LIN {X 0,Y 246.152,Z 600.24,A -85,B 0,C 180,E1 -19920.091,E2 -19920.091} C_VEL
LIN {X 0,Y 247.15,Z 576.037,A -85,B 0,C 180,E1 -19920.831,E2 -19920.831} C_VEL
LIN {X 0,Y 248.137,Z 547.926,A -85,B 0,C 180,E1 -19921.626,E2 -19921.626} C_VEL
LIN {X 0,Y 244.245,Z 525.026,A -85,B 0,C 180,E1 -19922.967,E2 -19922.967} C_VEL
LIN {X 0,Y 243.144,Z 521.008,A -85,B 0,C 180,E1 -19923.272,E2 -19923.272} C_VEL
LIN {X 0,Y 237.077,Z 506.902,A -85,B 0,C 180,E1 -19924.739,E2 -19924.739} C_VEL
LIN {X 0,Y 231.234,Z 495.155,A -85,B 0,C 180,E1 -19926.183,E2 -19926.183} C_VEL
LIN {X 0,Y 230.085,Z 492.253,A -85,B 0,C 180,E1 -19926.602,E2 -19926.602} C_VEL
LIN {X 0,Y 228.669,Z 486.217,A -85,B 0,C 180,E1 -19930.197,E2 -19930.197} C_VEL
LIN {X 0,Y 227.823,Z 482.666,A -85,B 0,C 180,E1 -19932.575,E2 -19932.575} C_VEL
LIN {X 0,Y 227.795,Z 482.606,A -85,B 0,C 180,E1 -19937.251,E2 -19937.251} C_VEL
LIN {X 0,Y 227.844,Z 482.598,A -85,B 0,C 180,E1 -19941.906,E2 -19941.906} C_VEL
LIN {X 0,Y 227.879,Z 482.572,A -85,B 0,C 180,E1 -19946.376,E2 -19946.376} C_VEL
LIN {X 0,Y 227.877,Z 482.596,A -85,B 0,C 180,E1 -19950.429,E2 -19950.429} C_VEL
LIN {X 0,Y 227.867,Z 482.569,A -85,B 0,C 180,E1 -19954.416,E2 -19954.416} C_VEL
LIN {X 0,Y 227.919,Z 482.587,A -85,B 0,C 180,E1 -19958.28,E2 -19958.28} C_VEL
LIN {X 0,Y 227.998,Z 482.563,A -85,B 0,C 180,E1 -19963.891,E2 -19963.891} C_VEL
LIN {X 0,Y 228.123,Z 482.528,A -85,B 0,C 180,E1 -19969.345,E2 -19969.345} C_VEL
LIN {X 0,Y 228.291,Z 482.521,A -85,B 0,C 180,E1 -19972.924,E2 -19972.924} C_VEL
LIN {X 0,Y 228.528,Z 482.492,A -85,B 0,C 180,E1 -19978.235,E2 -19978.235} C_VEL
LIN {X 0,Y 228.503,Z 482.481,A -85,B 0,C 180,E1 -19981.76,E2 -19981.76} C_VEL
LIN {X 0,Y 228.294,Z 482.536,A -85,B 0,C 180,E1 -19987.071,E2 -19987.071} C_VEL
LIN {X 0,Y 228.121,Z 482.525,A -85,B 0,C 180,E1 -19990.649,E2 -19990.649} C_VEL
LIN {X 0,Y 228.004,Z 482.577,A -85,B 0,C 180,E1 -19996.103,E2 -19996.103} C_VEL
LIN {X 0,Y 227.912,Z 482.579,A -85,B 0,C 180,E1 -20001.715,E2 -20001.715} C_VEL
LIN {X 0,Y 227.862,Z 482.571,A -85,B 0,C 180,E1 -20006.563,E2 -20006.563} C_VEL
LIN {X 0,Y 227.861,Z 482.597,A -85,B 0,C 180,E1 -20010.276,E2 -20010.276} C_VEL
LIN {X 0,Y 227.863,Z 482.578,A -85,B 0,C 180,E1 -20013.719,E2 -20013.719} C_VEL
LIN {X 0,Y 227.827,Z 482.608,A -85,B 0,C 180,E1 -20018.09,E2 -20018.09} C_VEL
LIN {X 0,Y 227.772,Z 482.608,A -85,B 0,C 180,E1 -20022.747,E2 -20022.747} C_VEL
LIN {X 0,Y 227.794,Z 482.578,A -85,B 0,C 180,E1 -20025.198,E2 -20025.198} C_VEL
LIN {X 0,Y 227.783,Z 482.557,A -85,B 0,C 180,E1 -20029.615,E2 -20029.615} C_VEL
LIN {X 0,Y 227.873,Z 482.738,A -85,B 0,C 180,E1 -20032.789,E2 -20032.789} C_VEL
LIN {X 0,Y 228.097,Z 483.675,A -85,B 0,C 180,E1 -20033.156,E2 -20033.156} C_VEL
LIN {X 0,Y 229.658,Z 486.481,A -85,B 0,C 180,E1 -20033.59,E2 -20033.59} C_VEL
LIN {X 0,Y 235.192,Z 495.686,A -85,B 0,C 180,E1 -20034.923,E2 -20034.923} C_VEL
LIN {X 0,Y 242.911,Z 509.793,A -85,B 0,C 180,E1 -20036.692,E2 -20036.692} C_VEL
LIN {X 0,Y 251.381,Z 526.173,A -85,B 0,C 180,E1 -20038.501,E2 -20038.501} C_VEL
LIN {X 0,Y 258.769,Z 537.403,A -85,B 0,C 180,E1 -20039.86,E2 -20039.86} C_VEL
LIN {X 0,Y 266.168,Z 546.904,A -85,B 0,C 180,E1 -20041.076,E2 -20041.076} C_VEL
LIN {X 0,Y 278.31,Z 560.203,A -85,B 0,C 180,E1 -20042.838,E2 -20042.838} C_VEL
LIN {X 0,Y 289.982,Z 571.118,A -85,B 0,C 180,E1 -20044.32,E2 -20044.32} C_VEL
LIN {X 0,Y 299.622,Z 579.319,A -85,B 0,C 180,E1 -20045.452,E2 -20045.452} C_VEL
LIN {X 0,Y 307.537,Z 585.808,A -85,B 0,C 180,E1 -20046.478,E2 -20046.478} C_VEL
LIN {X 0,Y 315.775,Z 592.173,A -85,B 0,C 180,E1 -20047.768,E2 -20047.768} C_VEL
LIN {X 0,Y 323.39,Z 597.842,A -85,B 0,C 180,E1 -20049.138,E2 -20049.138} C_VEL
LIN {X 0,Y 330.86,Z 603.38,A -85,B 0,C 180,E1 -20050.658,E2 -20050.658} C_VEL
LIN {X 0,Y 338.279,Z 608.514,A -85,B 0,C 180,E1 -20052.351,E2 -20052.351} C_VEL
LIN {X 0,Y 344.516,Z 613.086,A -85,B 0,C 180,E1 -20053.974,E2 -20053.974} C_VEL
LIN {X 0,Y 348.895,Z 616.008,A -85,B 0,C 180,E1 -20055.206,E2 -20055.206} C_VEL
LIN {X 0,Y 353.8,Z 618.948,A -85,B 0,C 180,E1 -20056.732,E2 -20056.732} C_VEL
LIN {X 0,Y 357.248,Z 621.232,A -85,B 0,C 180,E1 -20057.965,E2 -20057.965} C_VEL
LIN {X 0,Y 361.911,Z 624.66,A -85,B 0,C 180,E1 -20059.935,E2 -20059.935} C_VEL
LIN {X 0,Y 364.421,Z 626.158,A -85,B 0,C 180,E1 -20061.125,E2 -20061.125} C_VEL
LIN {X 0,Y 368.041,Z 628.101,A -85,B 0,C 180,E1 -20063.184,E2 -20063.184} C_VEL
LIN {X 0,Y 369.955,Z 628.948,A -85,B 0,C 180,E1 -20064.55,E2 -20064.55} C_VEL
LIN {X 0,Y 371.243,Z 629.373,A -85,B 0,C 180,E1 -20065.657,E2 -20065.657} C_VEL
LIN {X 0,Y 372.23,Z 629.672,A -85,B 0,C 180,E1 -20066.753,E2 -20066.753} C_VEL
LIN {X 0,Y 372.855,Z 630.069,A -85,B 0,C 180,E1 -20067.84,E2 -20067.84} C_VEL
LIN {X 0,Y 373.209,Z 630.352,A -85,B 0,C 180,E1 -20068.921,E2 -20068.921} C_VEL
LIN {X 0,Y 373.398,Z 630.248,A -85,B 0,C 180,E1 -20070,E2 -20070} C_VEL
LIN {X 0,Y 373.231,Z 630.289,A -85,B 0,C 180,E1 -20071.079,E2 -20071.079} C_VEL
LIN {X 0,Y 372.781,Z 630.004,A -85,B 0,C 180,E1 -20072.349,E2 -20072.349} C_VEL
LIN {X 0,Y 372.229,Z 629.672,A -85,B 0,C 180,E1 -20073.247,E2 -20073.247} C_VEL
LIN {X 0,Y 371.24,Z 629.386,A -85,B 0,C 180,E1 -20074.343,E2 -20074.343} C_VEL
LIN {X 0,Y 369.963,Z 628.952,A -85,B 0,C 180,E1 -20075.45,E2 -20075.45} C_VEL
LIN {X 0,Y 368.049,Z 628.078,A -85,B 0,C 180,E1 -20076.826,E2 -20076.826} C_VEL
LIN {X 0,Y 366.561,Z 627.405,A -85,B 0,C 180,E1 -20077.713,E2 -20077.713} C_VEL
LIN {X 0,Y 363.297,Z 625.502,A -85,B 0,C 180,E1 -20079.407,E2 -20079.407} C_VEL
LIN {X 0,Y 361.921,Z 624.674,A -85,B 0,C 180,E1 -20080.065,E2 -20080.065} C_VEL
LIN {X 0,Y 357.616,Z 621.526,A -85,B 0,C 180,E1 -20081.887,E2 -20081.887} C_VEL
LIN {X 0,Y 353.791,Z 618.959,A -85,B 0,C 180,E1 -20083.262,E2 -20083.262} C_VEL
LIN {X 0,Y 347.291,Z 614.974,A -85,B 0,C 180,E1 -20085.252,E2 -20085.252} C_VEL
LIN {X 0,Y 340.677,Z 610.221,A -85,B 0,C 180,E1 -20087.062,E2 -20087.062} C_VEL
LIN {X 0,Y 333.125,Z 605.057,A -85,B 0,C 180,E1 -20088.843,E2 -20088.843} C_VEL
LIN {X 0,Y 324.559,Z 598.647,A -85,B 0,C 180,E1 -20090.638,E2 -20090.638} C_VEL
LIN {X 0,Y 316.695,Z 592.953,A -85,B 0,C 180,E1 -20092.071,E2 -20092.071} C_VEL
LIN {X 0,Y 308.97,Z 586.887,A -85,B 0,C 180,E1 -20093.315,E2 -20093.315} C_VEL
LIN {X 0,Y 301.688,Z 581.017,A -85,B 0,C 180,E1 -20094.302,E2 -20094.302} C_VEL
LIN {X 0,Y 290.907,Z 571.969,A -85,B 0,C 180,E1 -20095.569,E2 -20095.569} C_VEL
LIN {X 0,Y 280.514,Z 562.3,A -85,B 0,C 180,E1 -20096.87,E2 -20096.87} C_VEL
LIN {X 0,Y 268.243,Z 549.356,A -85,B 0,C 180,E1 -20098.604,E2 -20098.604} C_VEL
LIN {X 0,Y 260.21,Z 539.392,A -85,B 0,C 180,E1 -20099.892,E2 -20099.892} C_VEL
LIN {X 0,Y 251.95,Z 527.134,A -85,B 0,C 180,E1 -20101.388,E2 -20101.388} C_VEL
LIN {X 0,Y 244.918,Z 513.819,A -85,B 0,C 180,E1 -20102.86,E2 -20102.86} C_VEL
LIN {X 0,Y 237.684,Z 500.018,A -85,B 0,C 180,E1 -20104.497,E2 -20104.497} C_VEL
LIN {X 0,Y 231.453,Z 489.468,A -85,B 0,C 180,E1 -20105.968,E2 -20105.968} C_VEL
LIN {X 0,Y 229.657,Z 486.509,A -85,B 0,C 180,E1 -20106.409,E2 -20106.409} C_VEL
LIN {X 0,Y 228.093,Z 483.698,A -85,B 0,C 180,E1 -20106.843,E2 -20106.843} C_VEL
LIN {X 0,Y 227.873,Z 482.743,A -85,B 0,C 180,E1 -20107.212,E2 -20107.212} C_VEL
LIN {X 0,Y 227.783,Z 482.557,A -85,B 0,C 180,E1 -20110.385,E2 -20110.385} C_VEL
LIN {X 0,Y 227.795,Z 482.588,A -85,B 0,C 180,E1 -20115.202,E2 -20115.202} C_VEL
LIN {X 0,Y 227.786,Z 482.59,A -85,B 0,C 180,E1 -20119.619,E2 -20119.619} C_VEL
LIN {X 0,Y 227.849,Z 482.584,A -85,B 0,C 180,E1 -20124.126,E2 -20124.126} C_VEL
LIN {X 0,Y 227.845,Z 482.605,A -85,B 0,C 180,E1 -20128.378,E2 -20128.378} C_VEL
LIN {X 0,Y 227.825,Z 482.572,A -85,B 0,C 180,E1 -20132.44,E2 -20132.44} C_VEL
LIN {X 0,Y 227.858,Z 482.603,A -85,B 0,C 180,E1 -20136.365,E2 -20136.365} C_VEL
LIN {X 0,Y 227.88,Z 482.559,A -85,B 0,C 180,E1 -20140.172,E2 -20140.172} C_VEL
LIN {X 0,Y 228.004,Z 482.577,A -85,B 0,C 180,E1 -20143.897,E2 -20143.897} C_VEL
LIN {X 0,Y 228.121,Z 482.525,A -85,B 0,C 180,E1 -20149.351,E2 -20149.351} C_VEL
LIN {X 0,Y 228.294,Z 482.536,A -85,B 0,C 180,E1 -20152.929,E2 -20152.929} C_VEL
LIN {X 0,Y 228.503,Z 482.481,A -85,B 0,C 180,E1 -20158.24,E2 -20158.24} C_VEL
LIN {X 0,Y 228.528,Z 482.492,A -85,B 0,C 180,E1 -20161.765,E2 -20161.765} C_VEL
LIN {X 0,Y 228.291,Z 482.521,A -85,B 0,C 180,E1 -20167.076,E2 -20167.076} C_VEL
LIN {X 0,Y 228.123,Z 482.528,A -85,B 0,C 180,E1 -20170.655,E2 -20170.655} C_VEL
LIN {X 0,Y 227.998,Z 482.563,A -85,B 0,C 180,E1 -20176.109,E2 -20176.109} C_VEL
LIN {X 0,Y 227.919,Z 482.587,A -85,B 0,C 180,E1 -20181.72,E2 -20181.72} C_VEL
LIN {X 0,Y 227.872,Z 482.564,A -85,B 0,C 180,E1 -20186.568,E2 -20186.568} C_VEL
LIN {X 0,Y 227.875,Z 482.601,A -85,B 0,C 180,E1 -20190.282,E2 -20190.282} C_VEL
LIN {X 0,Y 227.876,Z 482.572,A -85,B 0,C 180,E1 -20193.723,E2 -20193.723} C_VEL
LIN {X 0,Y 227.844,Z 482.598,A -85,B 0,C 180,E1 -20198.094,E2 -20198.094} C_VEL
LIN {X 0,Y 227.795,Z 482.606,A -85,B 0,C 180,E1 -20202.749,E2 -20202.749} C_VEL
LIN {X 0,Y 227.821,Z 482.677,A -85,B 0,C 180,E1 -20207.425,E2 -20207.425} C_VEL
LIN {X 0,Y 229.242,Z 488.495,A -85,B 0,C 180,E1 -20211.232,E2 -20211.232} C_VEL
LIN {X 0,Y 230.107,Z 492.26,A -85,B 0,C 180,E1 -20213.403,E2 -20213.403} C_VEL
LIN {X 0,Y 231.786,Z 496.084,A -85,B 0,C 180,E1 -20213.951,E2 -20213.951} C_VEL
LIN {X 0,Y 238.336,Z 509.677,A -85,B 0,C 180,E1 -20215.568,E2 -20215.568} C_VEL
LIN {X 0,Y 243.688,Z 522.323,A -85,B 0,C 180,E1 -20216.856,E2 -20216.856} C_VEL
LIN {X 0,Y 247.536,Z 543.646,A -85,B 0,C 180,E1 -20218.146,E2 -20218.146} C_VEL
LIN {X 0,Y 248.135,Z 549.551,A -85,B 0,C 180,E1 -20218.428,E2 -20218.428} C_VEL
LIN {X 0,Y 248.055,Z 551.394,A -85,B 0,C 180,E1 -20218.478,E2 -20218.478} C_VEL
LIN {X 0,Y 247.294,Z 555.318,A -85,B 0,C 180,E1 -20218.501,E2 -20218.501} C_VEL
LIN {X 0,Y 241.893,Z 567.619,A -85,B 0,C 180,E1 -20218.141,E2 -20218.141} C_VEL
LIN {X 0,Y 241.238,Z 571.533,A -85,B 0,C 180,E1 -20218.179,E2 -20218.179} C_VEL
LIN {X 0,Y 240.016,Z 599.524,A -85,B 0,C 180,E1 -20219.032,E2 -20219.032} C_VEL
LIN {X 0,Y 239.072,Z 609.938,A -85,B 0,C 180,E1 -20219.538,E2 -20219.538} C_VEL
LIN {X 0,Y 237.776,Z 619.744,A -85,B 0,C 180,E1 -20220.203,E2 -20220.203} C_VEL
LIN {X 0,Y 236.276,Z 629.543,A -85,B 0,C 180,E1 -20221.096,E2 -20221.096} C_VEL
LIN {X 0,Y 234.598,Z 638.308,A -85,B 0,C 180,E1 -20222.09,E2 -20222.09} C_VEL
LIN {X 0,Y 232.712,Z 647.03,A -85,B 0,C 180,E1 -20223.306,E2 -20223.306} C_VEL
LIN {X 0,Y 230.942,Z 654.441,A -85,B 0,C 180,E1 -20224.542,E2 -20224.542} C_VEL
LIN {X 0,Y 229.022,Z 661.859,A -85,B 0,C 180,E1 -20226.009,E2 -20226.009} C_VEL
LIN {X 0,Y 227.089,Z 669.094,A -85,B 0,C 180,E1 -20227.721,E2 -20227.721} C_VEL
LIN {X 0,Y 225.118,Z 676.649,A -85,B 0,C 180,E1 -20229.915,E2 -20229.915} C_VEL
LIN {X 0,Y 223.195,Z 682.958,A -85,B 0,C 180,E1 -20232.121,E2 -20232.121} C_VEL
LIN {X 0,Y 221.66,Z 688.231,A -85,B 0,C 180,E1 -20234.366,E2 -20234.366} C_VEL
LIN {X 0,Y 220.23,Z 693.327,A -85,B 0,C 180,E1 -20237.092,E2 -20237.092} C_VEL
LIN {X 0,Y 219.325,Z 697.296,A -85,B 0,C 180,E1 -20239.849,E2 -20239.849} C_VEL
LIN {X 0,Y 218.716,Z 700.234,A -85,B 0,C 180,E1 -20242.615,E2 -20242.615} C_VEL
LIN {X 0,Y 218.512,Z 701.738,A -85,B 0,C 180,E1 -20244.463,E2 -20244.463} C_VEL
LIN {X 0,Y 218.526,Z 703.271,A -85,B 0,C 180,E1 -20248.157,E2 -20248.157} C_VEL
LIN {X 0,Y 218.625,Z 703.554,A -85,B 0,C 180,E1 -20250,E2 -20250} C_VEL
LIN {X 0,Y 218.506,Z 702.672,A -85,B 0,C 180,E1 -20253.688,E2 -20253.688} C_VEL
LIN {X 0,Y 218.572,Z 701.74,A -85,B 0,C 180,E1 -20255.535,E2 -20255.535} C_VEL
LIN {X 0,Y 219.094,Z 698.386,A -85,B 0,C 180,E1 -20259.229,E2 -20259.229} C_VEL
LIN {X 0,Y 219.886,Z 694.756,A -85,B 0,C 180,E1 -20261.991,E2 -20261.991} C_VEL
LIN {X 0,Y 221.084,Z 690.02,A -85,B 0,C 180,E1 -20264.733,E2 -20264.733} C_VEL
LIN {X 0,Y 222.92,Z 684.052,A -85,B 0,C 180,E1 -20267.428,E2 -20267.428} C_VEL
LIN {X 0,Y 224.301,Z 679.271,A -85,B 0,C 180,E1 -20269.208,E2 -20269.208} C_VEL
LIN {X 0,Y 226.061,Z 673.153,A -85,B 0,C 180,E1 -20271.14,E2 -20271.14} C_VEL
LIN {X 0,Y 228.034,Z 665.56,A -85,B 0,C 180,E1 -20273.138,E2 -20273.138} C_VEL
LIN {X 0,Y 230.131,Z 657.736,A -85,B 0,C 180,E1 -20274.829,E2 -20274.829} C_VEL
LIN {X 0,Y 232.108,Z 649.654,A -85,B 0,C 180,E1 -20276.284,E2 -20276.284} C_VEL
LIN {X 0,Y 234.303,Z 639.898,A -85,B 0,C 180,E1 -20277.705,E2 -20277.705} C_VEL
LIN {X 0,Y 235.954,Z 631.511,A -85,B 0,C 180,E1 -20278.704,E2 -20278.704} C_VEL
LIN {X 0,Y 237.557,Z 621.005,A -85,B 0,C 180,E1 -20279.705,E2 -20279.705} C_VEL
LIN {X 0,Y 238.961,Z 610.702,A -85,B 0,C 180,E1 -20280.423,E2 -20280.423} C_VEL
LIN {X 0,Y 239.98,Z 600.72,A -85,B 0,C 180,E1 -20280.917,E2 -20280.917} C_VEL
LIN {X 0,Y 240.951,Z 579.375,A -85,B 0,C 180,E1 -20281.594,E2 -20281.594} C_VEL
LIN {X 0,Y 241.993,Z 548.404,A -85,B 0,C 180,E1 -20282.503,E2 -20282.503} C_VEL
LIN {X 0,Y 238.141,Z 525.634,A -85,B 0,C 180,E1 -20283.896,E2 -20283.896} C_VEL
LIN {X 0,Y 232.971,Z 512.992,A -85,B 0,C 180,E1 -20285.213,E2 -20285.213} C_VEL
LIN {X 0,Y 226.478,Z 499.636,A -85,B 0,C 180,E1 -20286.888,E2 -20286.888} C_VEL
LIN {X 0,Y 223.937,Z 494.745,A -85,B 0,C 180,E1 -20287.567,E2 -20287.567} C_VEL
LIN {X 0,Y 222.807,Z 492.019,A -85,B 0,C 180,E1 -20288.001,E2 -20288.001} C_VEL
LIN {X 0,Y 221.315,Z 485.957,A -85,B 0,C 180,E1 -20291.825,E2 -20291.825} C_VEL
LIN {X 0,Y 220.753,Z 483.553,A -85,B 0,C 180,E1 -20293.585,E2 -20293.585} C_VEL
LIN {X 0,Y 220.756,Z 483.487,A -85,B 0,C 180,E1 -20298.041,E2 -20298.041} C_VEL
LIN {X 0,Y 220.829,Z 483.479,A -85,B 0,C 180,E1 -20302.791,E2 -20302.791} C_VEL
LIN {X 0,Y 220.814,Z 483.457,A -85,B 0,C 180,E1 -20307.241,E2 -20307.241} C_VEL
LIN {X 0,Y 220.796,Z 483.46,A -85,B 0,C 180,E1 -20311.478,E2 -20311.478} C_VEL
LIN {X 0,Y 220.797,Z 483.464,A -85,B 0,C 180,E1 -20315.554,E2 -20315.554} C_VEL
LIN {X 0,Y 220.845,Z 483.449,A -85,B 0,C 180,E1 -20319.507,E2 -20319.507} C_VEL
LIN {X 0,Y 220.944,Z 483.431,A -85,B 0,C 180,E1 -20323.362,E2 -20323.362} C_VEL
LIN {X 0,Y 221.045,Z 483.413,A -85,B 0,C 180,E1 -20329,E2 -20329} C_VEL
LIN {X 0,Y 221.228,Z 483.396,A -85,B 0,C 180,E1 -20332.697,E2 -20332.697} C_VEL
LIN {X 0,Y 221.461,Z 483.372,A -85,B 0,C 180,E1 -20338.179,E2 -20338.179} C_VEL
LIN {X 0,Y 221.538,Z 483.341,A -85,B 0,C 180,E1 -20339.997,E2 -20339.997} C_VEL
LIN {X 0,Y 221.441,Z 483.36,A -85,B 0,C 180,E1 -20341.816,E2 -20341.816} C_VEL
LIN {X 0,Y 221.231,Z 483.411,A -85,B 0,C 180,E1 -20347.297,E2 -20347.297} C_VEL
LIN {X 0,Y 221.046,Z 483.407,A -85,B 0,C 180,E1 -20350.994,E2 -20350.994} C_VEL
LIN {X 0,Y 220.964,Z 483.446,A -85,B 0,C 180,E1 -20356.631,E2 -20356.631} C_VEL
LIN {X 0,Y 220.838,Z 483.44,A -85,B 0,C 180,E1 -20360.488,E2 -20360.488} C_VEL
LIN {X 0,Y 220.796,Z 483.478,A -85,B 0,C 180,E1 -20364.44,E2 -20364.44} C_VEL
LIN {X 0,Y 220.784,Z 483.453,A -85,B 0,C 180,E1 -20368.517,E2 -20368.517} C_VEL
LIN {X 0,Y 220.801,Z 483.468,A -85,B 0,C 180,E1 -20372.755,E2 -20372.755} C_VEL
LIN {X 0,Y 220.787,Z 483.483,A -85,B 0,C 180,E1 -20377.271,E2 -20377.271} C_VEL
LIN {X 0,Y 220.734,Z 483.474,A -85,B 0,C 180,E1 -20381.956,E2 -20381.956} C_VEL
LIN {X 0,Y 220.737,Z 483.447,A -85,B 0,C 180,E1 -20385.537,E2 -20385.537} C_VEL
LIN {X 0,Y 220.767,Z 483.444,A -85,B 0,C 180,E1 -20390.455,E2 -20390.455} C_VEL
LIN {X 0,Y 220.819,Z 483.766,A -85,B 0,C 180,E1 -20391.531,E2 -20391.531} C_VEL
LIN {X 0,Y 221.111,Z 484.873,A -85,B 0,C 180,E1 -20391.844,E2 -20391.844} C_VEL
LIN {X 0,Y 222.659,Z 487.488,A -85,B 0,C 180,E1 -20392.28,E2 -20392.28} C_VEL
LIN {X 0,Y 228.617,Z 497.051,A -85,B 0,C 180,E1 -20393.801,E2 -20393.801} C_VEL
LIN {X 0,Y 236.784,Z 511.74,A -85,B 0,C 180,E1 -20395.775,E2 -20395.775} C_VEL
LIN {X 0,Y 246.092,Z 530.036,A -85,B 0,C 180,E1 -20397.868,E2 -20397.868} C_VEL
LIN {X 0,Y 253.652,Z 541.708,A -85,B 0,C 180,E1 -20399.32,E2 -20399.32} C_VEL
LIN {X 0,Y 261.138,Z 551.49,A -85,B 0,C 180,E1 -20400.601,E2 -20400.601} C_VEL
LIN {X 0,Y 273.853,Z 565.494,A -85,B 0,C 180,E1 -20402.508,E2 -20402.508} C_VEL
LIN {X 0,Y 285.738,Z 576.669,A -85,B 0,C 180,E1 -20404.058,E2 -20404.058} C_VEL
LIN {X 0,Y 297.612,Z 586.737,A -85,B 0,C 180,E1 -20405.485,E2 -20405.485} C_VEL
LIN {X 0,Y 306.322,Z 593.716,A -85,B 0,C 180,E1 -20406.682,E2 -20406.682} C_VEL
LIN {X 0,Y 315.161,Z 600.552,A -85,B 0,C 180,E1 -20408.13,E2 -20408.13} C_VEL
LIN {X 0,Y 323.976,Z 606.917,A -85,B 0,C 180,E1 -20409.785,E2 -20409.785} C_VEL
LIN {X 0,Y 331.811,Z 612.657,A -85,B 0,C 180,E1 -20411.476,E2 -20411.476} C_VEL
LIN {X 0,Y 338.065,Z 616.973,A -85,B 0,C 180,E1 -20412.988,E2 -20412.988} C_VEL
LIN {X 0,Y 343.987,Z 621.179,A -85,B 0,C 180,E1 -20414.597,E2 -20414.597} C_VEL
LIN {X 0,Y 348.69,Z 624.181,A -85,B 0,C 180,E1 -20416.004,E2 -20416.004} C_VEL
LIN {X 0,Y 352.888,Z 626.57,A -85,B 0,C 180,E1 -20417.375,E2 -20417.375} C_VEL
LIN {X 0,Y 357.609,Z 630.137,A -85,B 0,C 180,E1 -20419.294,E2 -20419.294} C_VEL
LIN {X 0,Y 361.372,Z 632.529,A -85,B 0,C 180,E1 -20421.049,E2 -20421.049} C_VEL
LIN {X 0,Y 363.548,Z 633.753,A -85,B 0,C 180,E1 -20422.223,E2 -20422.223} C_VEL
LIN {X 0,Y 365.426,Z 634.705,A -85,B 0,C 180,E1 -20423.374,E2 -20423.374} C_VEL
LIN {X 0,Y 367.09,Z 635.43,A -85,B 0,C 180,E1 -20424.566,E2 -20424.566} C_VEL
LIN {X 0,Y 368.312,Z 635.847,A -85,B 0,C 180,E1 -20425.623,E2 -20425.623} C_VEL
LIN {X 0,Y 369.331,Z 636.134,A -85,B 0,C 180,E1 -20426.727,E2 -20426.727} C_VEL
LIN {X 0,Y 369.963,Z 636.524,A -85,B 0,C 180,E1 -20427.823,E2 -20427.823} C_VEL
LIN {X 0,Y 370.313,Z 636.808,A -85,B 0,C 180,E1 -20428.913,E2 -20428.913} C_VEL
LIN {X 0,Y 370.515,Z 636.708,A -85,B 0,C 180,E1 -20430,E2 -20430} C_VEL
LIN {X 0,Y 370.326,Z 636.764,A -85,B 0,C 180,E1 -20431.087,E2 -20431.087} C_VEL
LIN {X 0,Y 369.952,Z 636.522,A -85,B 0,C 180,E1 -20432.177,E2 -20432.177} C_VEL
LIN {X 0,Y 369.319,Z 636.128,A -85,B 0,C 180,E1 -20433.273,E2 -20433.273} C_VEL
LIN {X 0,Y 368.302,Z 635.842,A -85,B 0,C 180,E1 -20434.378,E2 -20434.378} C_VEL
LIN {X 0,Y 367.004,Z 635.393,A -85,B 0,C 180,E1 -20435.494,E2 -20435.494} C_VEL
LIN {X 0,Y 365.433,Z 634.696,A -85,B 0,C 180,E1 -20436.626,E2 -20436.626} C_VEL
LIN {X 0,Y 362.33,Z 633.119,A -85,B 0,C 180,E1 -20438.433,E2 -20438.433} C_VEL
LIN {X 0,Y 358.825,Z 631.037,A -85,B 0,C 180,E1 -20440.153,E2 -20440.153} C_VEL
LIN {X 0,Y 354.949,Z 628.21,A -85,B 0,C 180,E1 -20441.81,E2 -20441.81} C_VEL
LIN {X 0,Y 350.813,Z 625.364,A -85,B 0,C 180,E1 -20443.331,E2 -20443.331} C_VEL
LIN {X 0,Y 345.964,Z 622.467,A -85,B 0,C 180,E1 -20444.821,E2 -20444.821} C_VEL
LIN {X 0,Y 340.893,Z 619.012,A -85,B 0,C 180,E1 -20446.272,E2 -20446.272} C_VEL
LIN {X 0,Y 335.959,Z 615.335,A -85,B 0,C 180,E1 -20447.558,E2 -20447.558} C_VEL
LIN {X 0,Y 329.273,Z 610.899,A -85,B 0,C 180,E1 -20449.085,E2 -20449.085} C_VEL
LIN {X 0,Y 321.066,Z 604.786,A -85,B 0,C 180,E1 -20450.789,E2 -20450.789} C_VEL
LIN {X 0,Y 312.942,Z 598.863,A -85,B 0,C 180,E1 -20452.252,E2 -20452.252} C_VEL
LIN {X 0,Y 304.378,Z 592.212,A -85,B 0,C 180,E1 -20453.605,E2 -20453.605} C_VEL
LIN {X 0,Y 295.74,Z 585.188,A -85,B 0,C 180,E1 -20454.744,E2 -20454.744} C_VEL
LIN {X 0,Y 281.267,Z 572.743,A -85,B 0,C 180,E1 -20456.499,E2 -20456.499} C_VEL
LIN {X 0,Y 266.835,Z 558.072,A -85,B 0,C 180,E1 -20458.508,E2 -20458.508} C_VEL
LIN {X 0,Y 256.198,Z 545.289,A -85,B 0,C 180,E1 -20460.226,E2 -20460.226} C_VEL
LIN {X 0,Y 247.6,Z 532.566,A -85,B 0,C 180,E1 -20461.826,E2 -20461.826} C_VEL
LIN {X 0,Y 240.523,Z 519.383,A -85,B 0,C 180,E1 -20463.348,E2 -20463.348} C_VEL
LIN {X 0,Y 233.626,Z 505.89,A -85,B 0,C 180,E1 -20464.973,E2 -20464.973} C_VEL
LIN {X 0,Y 226.56,Z 493.674,A -85,B 0,C 180,E1 -20466.714,E2 -20466.714} C_VEL
LIN {X 0,Y 222.66,Z 487.466,A -85,B 0,C 180,E1 -20467.72,E2 -20467.72} C_VEL
LIN {X 0,Y 221.111,Z 484.873,A -85,B 0,C 180,E1 -20468.156,E2 -20468.156} C_VEL
LIN {X 0,Y 220.82,Z 483.706,A -85,B 0,C 180,E1 -20468.517,E2 -20468.517} C_VEL
LIN {X 0,Y 220.728,Z 483.423,A -85,B 0,C 180,E1 -20471.962,E2 -20471.962} C_VEL
LIN {X 0,Y 220.739,Z 483.474,A -85,B 0,C 180,E1 -20475.542,E2 -20475.542} C_VEL
LIN {X 0,Y 220.77,Z 483.469,A -85,B 0,C 180,E1 -20480.459,E2 -20480.459} C_VEL
LIN {X 0,Y 220.816,Z 483.479,A -85,B 0,C 180,E1 -20482.795,E2 -20482.795} C_VEL
LIN {X 0,Y 220.801,Z 483.468,A -85,B 0,C 180,E1 -20487.245,E2 -20487.245} C_VEL
LIN {X 0,Y 220.784,Z 483.453,A -85,B 0,C 180,E1 -20491.483,E2 -20491.483} C_VEL
LIN {X 0,Y 220.796,Z 483.478,A -85,B 0,C 180,E1 -20495.56,E2 -20495.56} C_VEL
LIN {X 0,Y 220.838,Z 483.44,A -85,B 0,C 180,E1 -20499.512,E2 -20499.512} C_VEL
LIN {X 0,Y 220.964,Z 483.446,A -85,B 0,C 180,E1 -20503.369,E2 -20503.369} C_VEL
LIN {X 0,Y 221.046,Z 483.407,A -85,B 0,C 180,E1 -20509.006,E2 -20509.006} C_VEL
LIN {X 0,Y 221.231,Z 483.411,A -85,B 0,C 180,E1 -20512.703,E2 -20512.703} C_VEL
LIN {X 0,Y 221.441,Z 483.36,A -85,B 0,C 180,E1 -20518.184,E2 -20518.184} C_VEL
LIN {X 0,Y 221.538,Z 483.341,A -85,B 0,C 180,E1 -20520.003,E2 -20520.003} C_VEL
LIN {X 0,Y 221.461,Z 483.372,A -85,B 0,C 180,E1 -20521.821,E2 -20521.821} C_VEL
LIN {X 0,Y 221.228,Z 483.396,A -85,B 0,C 180,E1 -20527.303,E2 -20527.303} C_VEL
LIN {X 0,Y 221.045,Z 483.413,A -85,B 0,C 180,E1 -20531,E2 -20531} C_VEL
LIN {X 0,Y 220.944,Z 483.431,A -85,B 0,C 180,E1 -20536.638,E2 -20536.638} C_VEL
LIN {X 0,Y 220.845,Z 483.449,A -85,B 0,C 180,E1 -20540.493,E2 -20540.493} C_VEL
LIN {X 0,Y 220.797,Z 483.464,A -85,B 0,C 180,E1 -20544.446,E2 -20544.446} C_VEL
LIN {X 0,Y 220.796,Z 483.46,A -85,B 0,C 180,E1 -20548.522,E2 -20548.522} C_VEL
LIN {X 0,Y 220.814,Z 483.457,A -85,B 0,C 180,E1 -20552.759,E2 -20552.759} C_VEL
LIN {X 0,Y 220.806,Z 483.482,A -85,B 0,C 180,E1 -20557.277,E2 -20557.277} C_VEL
LIN {X 0,Y 220.756,Z 483.487,A -85,B 0,C 180,E1 -20561.959,E2 -20561.959} C_VEL
LIN {X 0,Y 220.757,Z 483.626,A -85,B 0,C 180,E1 -20566.572,E2 -20566.572} C_VEL
LIN {X 0,Y 222.639,Z 491.302,A -85,B 0,C 180,E1 -20571.655,E2 -20571.655} C_VEL
LIN {X 0,Y 222.985,Z 492.547,A -85,B 0,C 180,E1 -20572.122,E2 -20572.122} C_VEL
LIN {X 0,Y 229.695,Z 506.052,A -85,B 0,C 180,E1 -20573.951,E2 -20573.951} C_VEL
LIN {X 0,Y 236.302,Z 520.801,A -85,B 0,C 180,E1 -20575.633,E2 -20575.633} C_VEL
LIN {X 0,Y 238.277,Z 526.324,A -85,B 0,C 180,E1 -20576.151,E2 -20576.151} C_VEL
LIN {X 0,Y 241.849,Z 547.149,A -85,B 0,C 180,E1 -20577.432,E2 -20577.432} C_VEL
LIN {X 0,Y 242.006,Z 552.1,A -85,B 0,C 180,E1 -20577.626,E2 -20577.626} C_VEL
LIN {X 0,Y 241.238,Z 571.533,A -85,B 0,C 180,E1 -20578.179,E2 -20578.179} C_VEL
LIN {X 0,Y 240.553,Z 577.376,A -85,B 0,C 180,E1 -20578.277,E2 -20578.277} C_VEL
LIN {X 0,Y 237.721,Z 586.874,A -85,B 0,C 180,E1 -20578.19,E2 -20578.19} C_VEL
LIN {X 0,Y 234.727,Z 596.356,A -85,B 0,C 180,E1 -20578.103,E2 -20578.103} C_VEL
LIN {X 0,Y 233.807,Z 602.18,A -85,B 0,C 180,E1 -20578.252,E2 -20578.252} C_VEL
LIN {X 0,Y 232.231,Z 615.762,A -85,B 0,C 180,E1 -20579.038,E2 -20579.038} C_VEL
LIN {X 0,Y 230.818,Z 625.412,A -85,B 0,C 180,E1 -20579.842,E2 -20579.842} C_VEL
LIN {X 0,Y 228.657,Z 636.521,A -85,B 0,C 180,E1 -20581.047,E2 -20581.047} C_VEL
LIN {X 0,Y 226.721,Z 645.521,A -85,B 0,C 180,E1 -20582.292,E2 -20582.292} C_VEL
LIN {X 0,Y 224.518,Z 654.244,A -85,B 0,C 180,E1 -20583.759,E2 -20583.759} C_VEL
LIN {X 0,Y 222.529,Z 661.662,A -85,B 0,C 180,E1 -20585.262,E2 -20585.262} C_VEL
LIN {X 0,Y 220.049,Z 670.458,A -85,B 0,C 180,E1 -20587.464,E2 -20587.464} C_VEL
LIN {X 0,Y 218.421,Z 676.452,A -85,B 0,C 180,E1 -20589.272,E2 -20589.272} C_VEL
LIN {X 0,Y 216.398,Z 682.76,A -85,B 0,C 180,E1 -20591.54,E2 -20591.54} C_VEL
LIN {X 0,Y 214.806,Z 688.034,A -85,B 0,C 180,E1 -20593.853,E2 -20593.853} C_VEL
LIN {X 0,Y 213.266,Z 693.129,A -85,B 0,C 180,E1 -20596.663,E2 -20596.663} C_VEL
LIN {X 0,Y 212.311,Z 697.099,A -85,B 0,C 180,E1 -20599.51,E2 -20599.51} C_VEL
LIN {X 0,Y 211.656,Z 700.038,A -85,B 0,C 180,E1 -20602.368,E2 -20602.368} C_VEL
LIN {X 0,Y 211.44,Z 701.542,A -85,B 0,C 180,E1 -20604.277,E2 -20604.277} C_VEL
LIN {X 0,Y 211.429,Z 703.075,A -85,B 0,C 180,E1 -20608.095,E2 -20608.095} C_VEL
LIN {X 0,Y 211.541,Z 703.358,A -85,B 0,C 180,E1 -20610,E2 -20610} C_VEL
LIN {X 0,Y 211.404,Z 702.475,A -85,B 0,C 180,E1 -20613.812,E2 -20613.812} C_VEL
LIN {X 0,Y 211.494,Z 701.543,A -85,B 0,C 180,E1 -20615.721,E2 -20615.721} C_VEL
LIN {X 0,Y 212.068,Z 698.19,A -85,B 0,C 180,E1 -20619.538,E2 -20619.538} C_VEL
LIN {X 0,Y 212.909,Z 694.559,A -85,B 0,C 180,E1 -20622.39,E2 -20622.39} C_VEL
LIN {X 0,Y 214.209,Z 689.824,A -85,B 0,C 180,E1 -20625.217,E2 -20625.217} C_VEL
LIN {X 0,Y 216.112,Z 683.854,A -85,B 0,C 180,E1 -20627.995,E2 -20627.995} C_VEL
LIN {X 0,Y 217.603,Z 679.075,A -85,B 0,C 180,E1 -20629.823,E2 -20629.823} C_VEL
LIN {X 0,Y 219.429,Z 672.84,A -85,B 0,C 180,E1 -20631.847,E2 -20631.847} C_VEL
LIN {X 0,Y 221.503,Z 665.363,A -85,B 0,C 180,E1 -20633.862,E2 -20633.862} C_VEL
LIN {X 0,Y 223.675,Z 657.539,A -85,B 0,C 180,E1 -20635.596,E2 -20635.596} C_VEL
LIN {X 0,Y 225.757,Z 649.458,A -85,B 0,C 180,E1 -20637.083,E2 -20637.083} C_VEL
LIN {X 0,Y 228.03,Z 639.701,A -85,B 0,C 180,E1 -20638.536,E2 -20638.536} C_VEL
LIN {X 0,Y 229.756,Z 631.315,A -85,B 0,C 180,E1 -20639.554,E2 -20639.554} C_VEL
LIN {X 0,Y 231.42,Z 620.808,A -85,B 0,C 180,E1 -20640.576,E2 -20640.576} C_VEL
LIN {X 0,Y 232.862,Z 610.674,A -85,B 0,C 180,E1 -20641.296,E2 -20641.296} C_VEL
LIN {X 0,Y 233.955,Z 600.047,A -85,B 0,C 180,E1 -20641.828,E2 -20641.828} C_VEL
LIN {X 0,Y 235.009,Z 576.988,A -85,B 0,C 180,E1 -20642.567,E2 -20642.567} C_VEL
LIN {X 0,Y 236.001,Z 549.279,A -85,B 0,C 180,E1 -20643.396,E2 -20643.396} C_VEL
LIN {X 0,Y 232.424,Z 527.995,A -85,B 0,C 180,E1 -20644.754,E2 -20644.754} C_VEL
LIN {X 0,Y 226.691,Z 514.279,A -85,B 0,C 180,E1 -20646.283,E2 -20646.283} C_VEL
LIN {X 0,Y 219.531,Z 499.708,A -85,B 0,C 180,E1 -20648.248,E2 -20648.248} C_VEL
LIN {X 0,Y 217.09,Z 495.214,A -85,B 0,C 180,E1 -20648.94,E2 -20648.94} C_VEL
LIN {X 0,Y 215.429,Z 491.711,A -85,B 0,C 180,E1 -20649.571,E2 -20649.571} C_VEL
LIN {X 0,Y 213.964,Z 485.519,A -85,B 0,C 180,E1 -20653.725,E2 -20653.725} C_VEL
LIN {X 0,Y 213.733,Z 484.415,A -85,B 0,C 180,E1 -20654.674,E2 -20654.674} C_VEL
LIN {X 0,Y 213.708,Z 484.352,A -85,B 0,C 180,E1 -20659.145,E2 -20659.145} C_VEL
LIN {X 0,Y 213.744,Z 484.354,A -85,B 0,C 180,E1 -20663.709,E2 -20663.709} C_VEL
LIN {X 0,Y 213.761,Z 484.348,A -85,B 0,C 180,E1 -20668.258,E2 -20668.258} C_VEL
LIN {X 0,Y 213.786,Z 484.32,A -85,B 0,C 180,E1 -20672.595,E2 -20672.595} C_VEL
LIN {X 0,Y 213.781,Z 484.353,A -85,B 0,C 180,E1 -20676.997,E2 -20676.997} C_VEL
LIN {X 0,Y 213.873,Z 484.304,A -85,B 0,C 180,E1 -20682.795,E2 -20682.795} C_VEL
LIN {X 0,Y 213.901,Z 484.335,A -85,B 0,C 180,E1 -20686.7,E2 -20686.7} C_VEL
LIN {X 0,Y 214.122,Z 484.263,A -85,B 0,C 180,E1 -20690.552,E2 -20690.552} C_VEL
LIN {X 0,Y 214.065,Z 484.313,A -85,B 0,C 180,E1 -20694.345,E2 -20694.345} C_VEL
LIN {X 0,Y 214.398,Z 484.251,A -85,B 0,C 180,E1 -20698.119,E2 -20698.119} C_VEL
LIN {X 0,Y 214.507,Z 484.216,A -85,B 0,C 180,E1 -20699.997,E2 -20699.997} C_VEL
LIN {X 0,Y 214.381,Z 484.239,A -85,B 0,C 180,E1 -20701.876,E2 -20701.876} C_VEL
LIN {X 0,Y 214.172,Z 484.286,A -85,B 0,C 180,E1 -20707.539,E2 -20707.539} C_VEL
LIN {X 0,Y 213.979,Z 484.289,A -85,B 0,C 180,E1 -20711.362,E2 -20711.362} C_VEL
LIN {X 0,Y 213.869,Z 484.345,A -85,B 0,C 180,E1 -20715.238,E2 -20715.238} C_VEL
LIN {X 0,Y 213.783,Z 484.312,A -85,B 0,C 180,E1 -20719.189,E2 -20719.189} C_VEL
LIN {X 0,Y 213.778,Z 484.356,A -85,B 0,C 180,E1 -20723.232,E2 -20723.232} C_VEL
LIN {X 0,Y 213.759,Z 484.323,A -85,B 0,C 180,E1 -20727.414,E2 -20727.414} C_VEL
LIN {X 0,Y 213.75,Z 484.359,A -85,B 0,C 180,E1 -20731.737,E2 -20731.737} C_VEL
LIN {X 0,Y 213.73,Z 484.346,A -85,B 0,C 180,E1 -20736.287,E2 -20736.287} C_VEL
LIN {X 0,Y 213.686,Z 484.346,A -85,B 0,C 180,E1 -20741.127,E2 -20741.127} C_VEL
LIN {X 0,Y 213.69,Z 484.367,A -85,B 0,C 180,E1 -20743.678,E2 -20743.678} C_VEL
LIN {X 0,Y 213.689,Z 484.31,A -85,B 0,C 180,E1 -20746.344,E2 -20746.344} C_VEL
LIN {X 0,Y 213.734,Z 484.435,A -85,B 0,C 180,E1 -20749.865,E2 -20749.865} C_VEL
LIN {X 0,Y 213.925,Z 485.28,A -85,B 0,C 180,E1 -20750.291,E2 -20750.291} C_VEL
LIN {X 0,Y 215.42,Z 488.138,A -85,B 0,C 180,E1 -20750.792,E2 -20750.792} C_VEL
LIN {X 0,Y 216.638,Z 489.798,A -85,B 0,C 180,E1 -20751.126,E2 -20751.126} C_VEL
LIN {X 0,Y 223.88,Z 501.507,A -85,B 0,C 180,E1 -20753.078,E2 -20753.078} C_VEL
LIN {X 0,Y 232.002,Z 516.356,A -85,B 0,C 180,E1 -20755.133,E2 -20755.133} C_VEL
LIN {X 0,Y 241.055,Z 534.316,A -85,B 0,C 180,E1 -20757.256,E2 -20757.256} C_VEL
LIN {X 0,Y 248.972,Z 546.63,A -85,B 0,C 180,E1 -20758.837,E2 -20758.837} C_VEL
LIN {X 0,Y 256.638,Z 556.661,A -85,B 0,C 180,E1 -20760.193,E2 -20760.193} C_VEL
LIN {X 0,Y 269.615,Z 570.999,A -85,B 0,C 180,E1 -20762.197,E2 -20762.197} C_VEL
LIN {X 0,Y 281.475,Z 582.203,A -85,B 0,C 180,E1 -20763.799,E2 -20763.799} C_VEL
LIN {X 0,Y 291.698,Z 590.966,A -85,B 0,C 180,E1 -20765.124,E2 -20765.124} C_VEL
LIN {X 0,Y 301.569,Z 598.963,A -85,B 0,C 180,E1 -20766.47,E2 -20766.47} C_VEL
LIN {X 0,Y 308.35,Z 604.228,A -85,B 0,C 180,E1 -20767.533,E2 -20767.533} C_VEL
LIN {X 0,Y 316.293,Z 610.071,A -85,B 0,C 180,E1 -20768.938,E2 -20768.938} C_VEL
LIN {X 0,Y 323.604,Z 615.509,A -85,B 0,C 180,E1 -20770.422,E2 -20770.422} C_VEL
LIN {X 0,Y 330.785,Z 620.439,A -85,B 0,C 180,E1 -20772.014,E2 -20772.014} C_VEL
LIN {X 0,Y 337.766,Z 625.502,A -85,B 0,C 180,E1 -20773.801,E2 -20773.801} C_VEL
LIN {X 0,Y 344.82,Z 630.114,A -85,B 0,C 180,E1 -20775.843,E2 -20775.843} C_VEL
LIN {X 0,Y 349.015,Z 632.535,A -85,B 0,C 180,E1 -20777.203,E2 -20777.203} C_VEL
LIN {X 0,Y 353.959,Z 636.192,A -85,B 0,C 180,E1 -20779.183,E2 -20779.183} C_VEL
LIN {X 0,Y 357.782,Z 638.638,A -85,B 0,C 180,E1 -20780.959,E2 -20780.959} C_VEL
LIN {X 0,Y 361.211,Z 640.535,A -85,B 0,C 180,E1 -20782.863,E2 -20782.863} C_VEL
LIN {X 0,Y 363.56,Z 641.592,A -85,B 0,C 180,E1 -20784.453,E2 -20784.453} C_VEL
LIN {X 0,Y 364.916,Z 642.097,A -85,B 0,C 180,E1 -20785.582,E2 -20785.582} C_VEL
LIN {X 0,Y 366.032,Z 642.419,A -85,B 0,C 180,E1 -20786.741,E2 -20786.741} C_VEL
LIN {X 0,Y 366.642,Z 642.795,A -85,B 0,C 180,E1 -20787.803,E2 -20787.803} C_VEL
LIN {X 0,Y 366.994,Z 643.08,A -85,B 0,C 180,E1 -20788.903,E2 -20788.903} C_VEL
LIN {X 0,Y 367.221,Z 642.975,A -85,B 0,C 180,E1 -20790,E2 -20790} C_VEL
LIN {X 0,Y 367.014,Z 643.03,A -85,B 0,C 180,E1 -20791.097,E2 -20791.097} C_VEL
LIN {X 0,Y 366.634,Z 642.786,A -85,B 0,C 180,E1 -20792.197,E2 -20792.197} C_VEL
LIN {X 0,Y 365.976,Z 642.404,A -85,B 0,C 180,E1 -20793.303,E2 -20793.303} C_VEL
LIN {X 0,Y 364.905,Z 642.081,A -85,B 0,C 180,E1 -20794.418,E2 -20794.418} C_VEL
LIN {X 0,Y 363.542,Z 641.587,A -85,B 0,C 180,E1 -20795.547,E2 -20795.547} C_VEL
LIN {X 0,Y 361.22,Z 640.538,A -85,B 0,C 180,E1 -20797.148,E2 -20797.148} C_VEL
LIN {X 0,Y 357.754,Z 638.66,A -85,B 0,C 180,E1 -20799.042,E2 -20799.042} C_VEL
LIN {X 0,Y 353.97,Z 636.232,A -85,B 0,C 180,E1 -20800.809,E2 -20800.809} C_VEL
LIN {X 0,Y 349.024,Z 632.568,A -85,B 0,C 180,E1 -20802.797,E2 -20802.797} C_VEL
LIN {X 0,Y 344.802,Z 630.097,A -85,B 0,C 180,E1 -20804.158,E2 -20804.158} C_VEL
LIN {X 0,Y 339.952,Z 627.005,A -85,B 0,C 180,E1 -20805.59,E2 -20805.59} C_VEL
LIN {X 0,Y 334.334,Z 622.957,A -85,B 0,C 180,E1 -20807.115,E2 -20807.115} C_VEL
LIN {X 0,Y 327.27,Z 618.096,A -85,B 0,C 180,E1 -20808.791,E2 -20808.791} C_VEL
LIN {X 0,Y 319.709,Z 612.501,A -85,B 0,C 180,E1 -20810.409,E2 -20810.409} C_VEL
LIN {X 0,Y 310.845,Z 606.165,A -85,B 0,C 180,E1 -20812.038,E2 -20812.038} C_VEL
LIN {X 0,Y 302.166,Z 599.416,A -85,B 0,C 180,E1 -20813.446,E2 -20813.446} C_VEL
LIN {X 0,Y 293.183,Z 592.167,A -85,B 0,C 180,E1 -20814.685,E2 -20814.685} C_VEL
LIN {X 0,Y 282.596,Z 583.246,A -85,B 0,C 180,E1 -20816.057,E2 -20816.057} C_VEL
LIN {X 0,Y 269.989,Z 571.375,A -85,B 0,C 180,E1 -20817.75,E2 -20817.75} C_VEL
LIN {X 0,Y 257.528,Z 557.68,A -85,B 0,C 180,E1 -20819.661,E2 -20819.661} C_VEL
LIN {X 0,Y 250.534,Z 548.817,A -85,B 0,C 180,E1 -20820.873,E2 -20820.873} C_VEL
LIN {X 0,Y 242.501,Z 536.755,A -85,B 0,C 180,E1 -20822.438,E2 -20822.438} C_VEL
LIN {X 0,Y 235.385,Z 523.354,A -85,B 0,C 180,E1 -20824.038,E2 -20824.038} C_VEL
LIN {X 0,Y 228.72,Z 510.168,A -85,B 0,C 180,E1 -20825.681,E2 -20825.681} C_VEL
LIN {X 0,Y 222.015,Z 498.404,A -85,B 0,C 180,E1 -20827.411,E2 -20827.411} C_VEL
LIN {X 0,Y 217.965,Z 492.01,A -85,B 0,C 180,E1 -20828.5,E2 -20828.5} C_VEL
LIN {X 0,Y 215.715,Z 488.432,A -85,B 0,C 180,E1 -20829.131,E2 -20829.131} C_VEL
LIN {X 0,Y 214.136,Z 485.963,A -85,B 0,C 180,E1 -20829.596,E2 -20829.596} C_VEL
LIN {X 0,Y 213.78,Z 484.637,A -85,B 0,C 180,E1 -20829.953,E2 -20829.953} C_VEL
LIN {X 0,Y 213.682,Z 484.303,A -85,B 0,C 180,E1 -20831.132,E2 -20831.132} C_VEL
LIN {X 0,Y 213.689,Z 484.31,A -85,B 0,C 180,E1 -20833.682,E2 -20833.682} C_VEL
LIN {X 0,Y 213.69,Z 484.367,A -85,B 0,C 180,E1 -20836.348,E2 -20836.348} C_VEL
LIN {X 0,Y 213.692,Z 484.362,A -85,B 0,C 180,E1 -20841.331,E2 -20841.331} C_VEL
LIN {X 0,Y 213.742,Z 484.335,A -85,B 0,C 180,E1 -20846.019,E2 -20846.019} C_VEL
LIN {X 0,Y 213.737,Z 484.344,A -85,B 0,C 180,E1 -20850.451,E2 -20850.451} C_VEL
LIN {X 0,Y 213.732,Z 484.345,A -85,B 0,C 180,E1 -20854.696,E2 -20854.696} C_VEL
LIN {X 0,Y 213.767,Z 484.329,A -85,B 0,C 180,E1 -20858.802,E2 -20858.802} C_VEL
LIN {X 0,Y 213.872,Z 484.318,A -85,B 0,C 180,E1 -20862.801,E2 -20862.801} C_VEL
LIN {X 0,Y 213.911,Z 484.328,A -85,B 0,C 180,E1 -20866.707,E2 -20866.707} C_VEL
LIN {X 0,Y 214.123,Z 484.267,A -85,B 0,C 180,E1 -20870.557,E2 -20870.557} C_VEL
LIN {X 0,Y 214.065,Z 484.321,A -85,B 0,C 180,E1 -20874.351,E2 -20874.351} C_VEL
LIN {X 0,Y 214.381,Z 484.239,A -85,B 0,C 180,E1 -20878.124,E2 -20878.124} C_VEL
LIN {X 0,Y 214.507,Z 484.216,A -85,B 0,C 180,E1 -20880.003,E2 -20880.003} C_VEL
LIN {X 0,Y 214.398,Z 484.251,A -85,B 0,C 180,E1 -20881.881,E2 -20881.881} C_VEL
LIN {X 0,Y 214.17,Z 484.27,A -85,B 0,C 180,E1 -20887.545,E2 -20887.545} C_VEL
LIN {X 0,Y 213.977,Z 484.298,A -85,B 0,C 180,E1 -20891.368,E2 -20891.368} C_VEL
LIN {X 0,Y 213.858,Z 484.334,A -85,B 0,C 180,E1 -20895.245,E2 -20895.245} C_VEL
LIN {X 0,Y 213.789,Z 484.311,A -85,B 0,C 180,E1 -20899.195,E2 -20899.195} C_VEL
LIN {X 0,Y 213.785,Z 484.353,A -85,B 0,C 180,E1 -20903.237,E2 -20903.237} C_VEL
LIN {X 0,Y 213.769,Z 484.322,A -85,B 0,C 180,E1 -20907.42,E2 -20907.42} C_VEL
LIN {X 0,Y 213.761,Z 484.348,A -85,B 0,C 180,E1 -20911.742,E2 -20911.742} C_VEL
LIN {X 0,Y 213.744,Z 484.354,A -85,B 0,C 180,E1 -20916.291,E2 -20916.291} C_VEL
LIN {X 0,Y 213.704,Z 484.355,A -85,B 0,C 180,E1 -20921.13,E2 -20921.13} C_VEL
LIN {X 0,Y 213.739,Z 484.469,A -85,B 0,C 180,E1 -20925.492,E2 -20925.492} C_VEL
LIN {X 0,Y 215.269,Z 491.109,A -85,B 0,C 180,E1 -20930.117,E2 -20930.117} C_VEL
LIN {X 0,Y 215.578,Z 492.161,A -85,B 0,C 180,E1 -20930.564,E2 -20930.564} C_VEL
LIN {X 0,Y 220.921,Z 502.386,A -85,B 0,C 180,E1 -20932.142,E2 -20932.142} C_VEL
LIN {X 0,Y 227.676,Z 516.514,A -85,B 0,C 180,E1 -20933.983,E2 -20933.983} C_VEL
LIN {X 0,Y 232.525,Z 528.349,A -85,B 0,C 180,E1 -20935.276,E2 -20935.276} C_VEL
LIN {X 0,Y 236.055,Z 549.768,A -85,B 0,C 180,E1 -20936.63,E2 -20936.63} C_VEL
LIN {X 0,Y 234.091,Z 597.885,A -85,B 0,C 180,E1 -20938.084,E2 -20938.084} C_VEL
LIN {X 0,Y 233.807,Z 602.18,A -85,B 0,C 180,E1 -20938.252,E2 -20938.252} C_VEL
LIN {X 0,Y 232.788,Z 607.931,A -85,B 0,C 180,E1 -20938.44,E2 -20938.44} C_VEL
LIN {X 0,Y 229.221,Z 617.093,A -85,B 0,C 180,E1 -20938.7,E2 -20938.7} C_VEL
LIN {X 0,Y 225.135,Z 626.023,A -85,B 0,C 180,E1 -20939.093,E2 -20939.093} C_VEL
LIN {X 0,Y 223.529,Z 631.417,A -85,B 0,C 180,E1 -20939.577,E2 -20939.577} C_VEL
LIN {X 0,Y 220.779,Z 644.012,A -85,B 0,C 180,E1 -20941.219,E2 -20941.219} C_VEL
LIN {X 0,Y 218.143,Z 654.047,A -85,B 0,C 180,E1 -20942.931,E2 -20942.931} C_VEL
LIN {X 0,Y 216.098,Z 661.466,A -85,B 0,C 180,E1 -20944.474,E2 -20944.474} C_VEL
LIN {X 0,Y 213.479,Z 670.261,A -85,B 0,C 180,E1 -20946.731,E2 -20946.731} C_VEL
LIN {X 0,Y 211.76,Z 676.255,A -85,B 0,C 180,E1 -20948.588,E2 -20948.588} C_VEL
LIN {X 0,Y 209.644,Z 682.563,A -85,B 0,C 180,E1 -20950.922,E2 -20950.922} C_VEL
LIN {X 0,Y 207.965,Z 687.837,A -85,B 0,C 180,E1 -20953.307,E2 -20953.307} C_VEL
LIN {X 0,Y 206.319,Z 692.931,A -85,B 0,C 180,E1 -20956.205,E2 -20956.205} C_VEL
LIN {X 0,Y 205.289,Z 696.902,A -85,B 0,C 180,E1 -20959.147,E2 -20959.147} C_VEL
LIN {X 0,Y 204.618,Z 699.841,A -85,B 0,C 180,E1 -20962.103,E2 -20962.103} C_VEL
LIN {X 0,Y 204.365,Z 701.345,A -85,B 0,C 180,E1 -20964.078,E2 -20964.078} C_VEL
LIN {X 0,Y 204.333,Z 702.879,A -85,B 0,C 180,E1 -20968.029,E2 -20968.029} C_VEL
LIN {X 0,Y 204.441,Z 703.162,A -85,B 0,C 180,E1 -20970,E2 -20970} C_VEL
LIN {X 0,Y 204.304,Z 702.278,A -85,B 0,C 180,E1 -20973.945,E2 -20973.945} C_VEL
LIN {X 0,Y 204.401,Z 701.346,A -85,B 0,C 180,E1 -20975.921,E2 -20975.921} C_VEL
LIN {X 0,Y 205.059,Z 697.993,A -85,B 0,C 180,E1 -20979.867,E2 -20979.867} C_VEL
LIN {X 0,Y 205.947,Z 694.361,A -85,B 0,C 180,E1 -20982.815,E2 -20982.815} C_VEL
LIN {X 0,Y 207.354,Z 689.627,A -85,B 0,C 180,E1 -20985.733,E2 -20985.733} C_VEL
LIN {X 0,Y 209.312,Z 683.656,A -85,B 0,C 180,E1 -20988.601,E2 -20988.601} C_VEL
LIN {X 0,Y 211.333,Z 677.566,A -85,B 0,C 180,E1 -20990.946,E2 -20990.946} C_VEL
LIN {X 0,Y 213.493,Z 670.261,A -85,B 0,C 180,E1 -20993.268,E2 -20993.268} C_VEL
LIN {X 0,Y 216.111,Z 661.467,A -85,B 0,C 180,E1 -20995.524,E2 -20995.524} C_VEL
LIN {X 0,Y 219.141,Z 650.574,A -85,B 0,C 180,E1 -20997.711,E2 -20997.711} C_VEL
LIN {X 0,Y 221.487,Z 641.095,A -85,B 0,C 180,E1 -20999.2,E2 -20999.2} C_VEL
LIN {X 0,Y 223.602,Z 631.119,A -85,B 0,C 180,E1 -21000.452,E2 -21000.452} C_VEL
LIN {X 0,Y 225.346,Z 620.612,A -85,B 0,C 180,E1 -21001.492,E2 -21001.492} C_VEL
LIN {X 0,Y 226.917,Z 609.946,A -85,B 0,C 180,E1 -21002.254,E2 -21002.254} C_VEL
LIN {X 0,Y 228.007,Z 599.469,A -85,B 0,C 180,E1 -21002.78,E2 -21002.78} C_VEL
LIN {X 0,Y 229.159,Z 574.865,A -85,B 0,C 180,E1 -21003.577,E2 -21003.577} C_VEL
LIN {X 0,Y 230.074,Z 550.288,A -85,B 0,C 180,E1 -21004.33,E2 -21004.33} C_VEL
LIN {X 0,Y 226.775,Z 530.579,A -85,B 0,C 180,E1 -21005.645,E2 -21005.645} C_VEL
LIN {X 0,Y 221.04,Z 516.776,A -85,B 0,C 180,E1 -21007.259,E2 -21007.259} C_VEL
LIN {X 0,Y 213.119,Z 500.702,A -85,B 0,C 180,E1 -21009.568,E2 -21009.568} C_VEL
LIN {X 0,Y 209.757,Z 495.029,A -85,B 0,C 180,E1 -21010.575,E2 -21010.575} C_VEL
LIN {X 0,Y 208.183,Z 491.633,A -85,B 0,C 180,E1 -21011.183,E2 -21011.183} C_VEL
LIN {X 0,Y 207.301,Z 488.073,A -85,B 0,C 180,E1 -21013.575,E2 -21013.575} C_VEL
LIN {X 0,Y 206.692,Z 485.301,A -85,B 0,C 180,E1 -21015.738,E2 -21015.738} C_VEL
LIN {X 0,Y 206.652,Z 485.226,A -85,B 0,C 180,E1 -21019.743,E2 -21019.743} C_VEL
LIN {X 0,Y 206.703,Z 485.216,A -85,B 0,C 180,E1 -21024.686,E2 -21024.686} C_VEL
LIN {X 0,Y 206.698,Z 485.238,A -85,B 0,C 180,E1 -21029.332,E2 -21029.332} C_VEL
LIN {X 0,Y 206.679,Z 485.202,A -85,B 0,C 180,E1 -21033.762,E2 -21033.762} C_VEL
LIN {X 0,Y 206.708,Z 485.23,A -85,B 0,C 180,E1 -21038.035,E2 -21038.035} C_VEL
LIN {X 0,Y 206.804,Z 485.179,A -85,B 0,C 180,E1 -21042.188,E2 -21042.188} C_VEL
LIN {X 0,Y 206.843,Z 485.217,A -85,B 0,C 180,E1 -21046.238,E2 -21046.238} C_VEL
LIN {X 0,Y 207.071,Z 485.141,A -85,B 0,C 180,E1 -21050.227,E2 -21050.227} C_VEL
LIN {X 0,Y 207.029,Z 485.188,A -85,B 0,C 180,E1 -21054.152,E2 -21054.152} C_VEL
LIN {X 0,Y 207.338,Z 485.13,A -85,B 0,C 180,E1 -21058.055,E2 -21058.055} C_VEL
LIN {X 0,Y 207.474,Z 485.091,A -85,B 0,C 180,E1 -21059.997,E2 -21059.997} C_VEL
LIN {X 0,Y 207.031,Z 485.187,A -85,B 0,C 180,E1 -21063.89,E2 -21063.89} C_VEL
LIN {X 0,Y 207.117,Z 485.158,A -85,B 0,C 180,E1 -21067.798,E2 -21067.798} C_VEL
LIN {X 0,Y 206.899,Z 485.174,A -85,B 0,C 180,E1 -21071.757,E2 -21071.757} C_VEL
LIN {X 0,Y 206.801,Z 485.22,A -85,B 0,C 180,E1 -21075.773,E2 -21075.773} C_VEL
LIN {X 0,Y 206.703,Z 485.195,A -85,B 0,C 180,E1 -21079.874,E2 -21079.874} C_VEL
LIN {X 0,Y 206.691,Z 485.237,A -85,B 0,C 180,E1 -21084.078,E2 -21084.078} C_VEL
LIN {X 0,Y 206.67,Z 485.209,A -85,B 0,C 180,E1 -21088.426,E2 -21088.426} C_VEL
LIN {X 0,Y 206.684,Z 485.222,A -85,B 0,C 180,E1 -21092.956,E2 -21092.956} C_VEL
LIN {X 0,Y 206.691,Z 485.213,A -85,B 0,C 180,E1 -21095.309,E2 -21095.309} C_VEL
LIN {X 0,Y 206.635,Z 485.224,A -85,B 0,C 180,E1 -21100.253,E2 -21100.253} C_VEL
LIN {X 0,Y 206.618,Z 485.228,A -85,B 0,C 180,E1 -21104.415,E2 -21104.415} C_VEL
LIN {X 0,Y 206.648,Z 485.344,A -85,B 0,C 180,E1 -21108.244,E2 -21108.244} C_VEL
LIN {X 0,Y 206.903,Z 486.36,A -85,B 0,C 180,E1 -21108.712,E2 -21108.712} C_VEL
LIN {X 0,Y 208.45,Z 489.11,A -85,B 0,C 180,E1 -21109.244,E2 -21109.244} C_VEL
LIN {X 0,Y 209.555,Z 490.436,A -85,B 0,C 180,E1 -21109.564,E2 -21109.564} C_VEL
LIN {X 0,Y 218.759,Z 505.15,A -85,B 0,C 180,E1 -21112.205,E2 -21112.205} C_VEL
LIN {X 0,Y 227.037,Z 520.521,A -85,B 0,C 180,E1 -21114.408,E2 -21114.408} C_VEL
LIN {X 0,Y 235.798,Z 538.158,A -85,B 0,C 180,E1 -21116.563,E2 -21116.563} C_VEL
LIN {X 0,Y 243.772,Z 550.755,A -85,B 0,C 180,E1 -21118.23,E2 -21118.23} C_VEL
LIN {X 0,Y 251.969,Z 561.614,A -85,B 0,C 180,E1 -21119.738,E2 -21119.738} C_VEL
LIN {X 0,Y 265.065,Z 576.18,A -85,B 0,C 180,E1 -21121.829,E2 -21121.829} C_VEL
LIN {X 0,Y 277.167,Z 587.721,A -85,B 0,C 180,E1 -21123.554,E2 -21123.554} C_VEL
LIN {X 0,Y 287.545,Z 596.696,A -85,B 0,C 180,E1 -21125.036,E2 -21125.036} C_VEL
LIN {X 0,Y 298.588,Z 605.607,A -85,B 0,C 180,E1 -21126.623,E2 -21126.623} C_VEL
LIN {X 0,Y 307.004,Z 612.112,A -85,B 0,C 180,E1 -21127.985,E2 -21127.985} C_VEL
LIN {X 0,Y 315.172,Z 617.948,A -85,B 0,C 180,E1 -21129.473,E2 -21129.473} C_VEL
LIN {X 0,Y 321.802,Z 622.96,A -85,B 0,C 180,E1 -21130.878,E2 -21130.878} C_VEL
LIN {X 0,Y 327.568,Z 626.787,A -85,B 0,C 180,E1 -21132.172,E2 -21132.172} C_VEL
LIN {X 0,Y 335.243,Z 632.38,A -85,B 0,C 180,E1 -21134.185,E2 -21134.185} C_VEL
LIN {X 0,Y 340.735,Z 635.909,A -85,B 0,C 180,E1 -21135.784,E2 -21135.784} C_VEL
LIN {X 0,Y 345.671,Z 638.861,A -85,B 0,C 180,E1 -21137.387,E2 -21137.387} C_VEL
LIN {X 0,Y 350.415,Z 642.366,A -85,B 0,C 180,E1 -21139.33,E2 -21139.33} C_VEL
LIN {X 0,Y 355.175,Z 645.311,A -85,B 0,C 180,E1 -21141.621,E2 -21141.621} C_VEL
LIN {X 0,Y 357.964,Z 646.77,A -85,B 0,C 180,E1 -21143.235,E2 -21143.235} C_VEL
LIN {X 0,Y 359.98,Z 647.668,A -85,B 0,C 180,E1 -21144.651,E2 -21144.651} C_VEL
LIN {X 0,Y 362.141,Z 648.357,A -85,B 0,C 180,E1 -21146.662,E2 -21146.662} C_VEL
LIN {X 0,Y 362.811,Z 648.745,A -85,B 0,C 180,E1 -21147.78,E2 -21147.78} C_VEL
LIN {X 0,Y 363.156,Z 649.048,A -85,B 0,C 180,E1 -21148.891,E2 -21148.891} C_VEL
LIN {X 0,Y 363.409,Z 648.945,A -85,B 0,C 180,E1 -21150,E2 -21150} C_VEL
LIN {X 0,Y 363.183,Z 648.992,A -85,B 0,C 180,E1 -21151.109,E2 -21151.109} C_VEL
LIN {X 0,Y 362.785,Z 648.753,A -85,B 0,C 180,E1 -21152.22,E2 -21152.22} C_VEL
LIN {X 0,Y 362.115,Z 648.354,A -85,B 0,C 180,E1 -21153.338,E2 -21153.338} C_VEL
LIN {X 0,Y 359.976,Z 647.658,A -85,B 0,C 180,E1 -21155.342,E2 -21155.342} C_VEL
LIN {X 0,Y 357.954,Z 646.75,A -85,B 0,C 180,E1 -21156.765,E2 -21156.765} C_VEL
LIN {X 0,Y 355.175,Z 645.362,A -85,B 0,C 180,E1 -21158.378,E2 -21158.378} C_VEL
LIN {X 0,Y 350.402,Z 642.397,A -85,B 0,C 180,E1 -21160.659,E2 -21160.659} C_VEL
LIN {X 0,Y 345.659,Z 638.855,A -85,B 0,C 180,E1 -21162.604,E2 -21162.604} C_VEL
LIN {X 0,Y 340.281,Z 635.631,A -85,B 0,C 180,E1 -21164.35,E2 -21164.35} C_VEL
LIN {X 0,Y 333.092,Z 630.823,A -85,B 0,C 180,E1 -21166.407,E2 -21166.407} C_VEL
LIN {X 0,Y 327.611,Z 626.798,A -85,B 0,C 180,E1 -21167.828,E2 -21167.828} C_VEL
LIN {X 0,Y 320.439,Z 621.923,A -85,B 0,C 180,E1 -21169.43,E2 -21169.43} C_VEL
LIN {X 0,Y 313.581,Z 616.808,A -85,B 0,C 180,E1 -21170.834,E2 -21170.834} C_VEL
LIN {X 0,Y 305.625,Z 611.072,A -85,B 0,C 180,E1 -21172.253,E2 -21172.253} C_VEL
LIN {X 0,Y 296.882,Z 604.28,A -85,B 0,C 180,E1 -21173.628,E2 -21173.628} C_VEL
LIN {X 0,Y 282.084,Z 592.202,A -85,B 0,C 180,E1 -21175.741,E2 -21175.741} C_VEL
LIN {X 0,Y 269.466,Z 580.556,A -85,B 0,C 180,E1 -21177.537,E2 -21177.537} C_VEL
LIN {X 0,Y 255.331,Z 565.63,A -85,B 0,C 180,E1 -21179.691,E2 -21179.691} C_VEL
LIN {X 0,Y 246.039,Z 553.986,A -85,B 0,C 180,E1 -21181.333,E2 -21181.333} C_VEL
LIN {X 0,Y 237.476,Z 541.023,A -85,B 0,C 180,E1 -21183.067,E2 -21183.067} C_VEL
LIN {X 0,Y 230.363,Z 527.476,A -85,B 0,C 180,E1 -21184.738,E2 -21184.738} C_VEL
LIN {X 0,Y 223.932,Z 514.575,A -85,B 0,C 180,E1 -21186.399,E2 -21186.399} C_VEL
LIN {X 0,Y 216.425,Z 501.25,A -85,B 0,C 180,E1 -21188.441,E2 -21188.441} C_VEL
LIN {X 0,Y 211.089,Z 493.041,A -85,B 0,C 180,E1 -21189.966,E2 -21189.966} C_VEL
LIN {X 0,Y 208.823,Z 489.482,A -85,B 0,C 180,E1 -21190.651,E2 -21190.651} C_VEL
LIN {X 0,Y 207.082,Z 486.862,A -85,B 0,C 180,E1 -21191.2,E2 -21191.2} C_VEL
LIN {X 0,Y 206.673,Z 485.554,A -85,B 0,C 180,E1 -21191.578,E2 -21191.578} C_VEL
LIN {X 0,Y 206.605,Z 485.183,A -85,B 0,C 180,E1 -21192.869,E2 -21192.869} C_VEL
LIN {X 0,Y 206.607,Z 485.244,A -85,B 0,C 180,E1 -21197.136,E2 -21197.136} C_VEL
LIN {X 0,Y 206.66,Z 485.239,A -85,B 0,C 180,E1 -21201.459,E2 -21201.459} C_VEL
LIN {X 0,Y 206.691,Z 485.213,A -85,B 0,C 180,E1 -21204.691,E2 -21204.691} C_VEL
LIN {X 0,Y 206.686,Z 485.238,A -85,B 0,C 180,E1 -21209.337,E2 -21209.337} C_VEL
LIN {X 0,Y 206.664,Z 485.212,A -85,B 0,C 180,E1 -21213.766,E2 -21213.766} C_VEL
LIN {X 0,Y 206.706,Z 485.221,A -85,B 0,C 180,E1 -21218.041,E2 -21218.041} C_VEL
LIN {X 0,Y 206.797,Z 485.19,A -85,B 0,C 180,E1 -21222.193,E2 -21222.193} C_VEL
LIN {X 0,Y 206.852,Z 485.213,A -85,B 0,C 180,E1 -21226.245,E2 -21226.245} C_VEL
LIN {X 0,Y 207.069,Z 485.143,A -85,B 0,C 180,E1 -21230.233,E2 -21230.233} C_VEL
LIN {X 0,Y 207.029,Z 485.196,A -85,B 0,C 180,E1 -21234.158,E2 -21234.158} C_VEL
LIN {X 0,Y 207.323,Z 485.118,A -85,B 0,C 180,E1 -21238.06,E2 -21238.06} C_VEL
LIN {X 0,Y 207.474,Z 485.091,A -85,B 0,C 180,E1 -21240.003,E2 -21240.003} C_VEL
LIN {X 0,Y 207.338,Z 485.13,A -85,B 0,C 180,E1 -21241.945,E2 -21241.945} C_VEL
LIN {X 0,Y 207.115,Z 485.144,A -85,B 0,C 180,E1 -21247.804,E2 -21247.804} C_VEL
LIN {X 0,Y 206.896,Z 485.185,A -85,B 0,C 180,E1 -21251.763,E2 -21251.763} C_VEL
LIN {X 0,Y 206.793,Z 485.206,A -85,B 0,C 180,E1 -21255.779,E2 -21255.779} C_VEL
LIN {X 0,Y 206.709,Z 485.198,A -85,B 0,C 180,E1 -21259.879,E2 -21259.879} C_VEL
LIN {X 0,Y 206.697,Z 485.224,A -85,B 0,C 180,E1 -21264.083,E2 -21264.083} C_VEL
LIN {X 0,Y 206.681,Z 485.214,A -85,B 0,C 180,E1 -21268.431,E2 -21268.431} C_VEL
LIN {X 0,Y 206.696,Z 485.212,A -85,B 0,C 180,E1 -21272.961,E2 -21272.961} C_VEL
LIN {X 0,Y 206.672,Z 485.238,A -85,B 0,C 180,E1 -21277.745,E2 -21277.745} C_VEL
LIN {X 0,Y 206.637,Z 485.24,A -85,B 0,C 180,E1 -21281.562,E2 -21281.562} C_VEL
LIN {X 0,Y 206.689,Z 485.435,A -85,B 0,C 180,E1 -21284.435,E2 -21284.435} C_VEL
LIN {X 0,Y 208.102,Z 491.413,A -85,B 0,C 180,E1 -21288.718,E2 -21288.718} C_VEL
LIN {X 0,Y 208.878,Z 493.426,A -85,B 0,C 180,E1 -21289.148,E2 -21289.148} C_VEL
LIN {X 0,Y 213.565,Z 501.53,A -85,B 0,C 180,E1 -21290.566,E2 -21290.566} C_VEL
LIN {X 0,Y 220.145,Z 514.995,A -85,B 0,C 180,E1 -21292.494,E2 -21292.494} C_VEL
LIN {X 0,Y 225.874,Z 528.25,A -85,B 0,C 180,E1 -21294.103,E2 -21294.103} C_VEL
LIN {X 0,Y 227.034,Z 531.555,A -85,B 0,C 180,E1 -21294.439,E2 -21294.439} C_VEL
LIN {X 0,Y 230.166,Z 551.224,A -85,B 0,C 180,E1 -21295.72,E2 -21295.72} C_VEL
LIN {X 0,Y 228.041,Z 598.404,A -85,B 0,C 180,E1 -21297.17,E2 -21297.17} C_VEL
LIN {X 0,Y 227.086,Z 608.517,A -85,B 0,C 180,E1 -21297.664,E2 -21297.664} C_VEL
LIN {X 0,Y 225.782,Z 618.09,A -85,B 0,C 180,E1 -21298.314,E2 -21298.314} C_VEL
LIN {X 0,Y 224.346,Z 627.184,A -85,B 0,C 180,E1 -21299.138,E2 -21299.138} C_VEL
LIN {X 0,Y 223.529,Z 631.417,A -85,B 0,C 180,E1 -21299.577,E2 -21299.577} C_VEL
LIN {X 0,Y 221.777,Z 636.7,A -85,B 0,C 180,E1 -21300.094,E2 -21300.094} C_VEL
LIN {X 0,Y 217.307,Z 644.965,A -85,B 0,C 180,E1 -21300.922,E2 -21300.922} C_VEL
LIN {X 0,Y 212.747,Z 652.983,A -85,B 0,C 180,E1 -21301.961,E2 -21301.961} C_VEL
LIN {X 0,Y 210.857,Z 657.474,A -85,B 0,C 180,E1 -21302.803,E2 -21302.803} C_VEL
LIN {X 0,Y 207.985,Z 666.819,A -85,B 0,C 180,E1 -21305.015,E2 -21305.015} C_VEL
LIN {X 0,Y 205.126,Z 676.057,A -85,B 0,C 180,E1 -21307.86,E2 -21307.86} C_VEL
LIN {X 0,Y 202.928,Z 682.366,A -85,B 0,C 180,E1 -21310.265,E2 -21310.265} C_VEL
LIN {X 0,Y 201.15,Z 687.64,A -85,B 0,C 180,E1 -21312.724,E2 -21312.724} C_VEL
LIN {X 0,Y 199.392,Z 692.734,A -85,B 0,C 180,E1 -21315.716,E2 -21315.716} C_VEL
LIN {X 0,Y 198.279,Z 696.704,A -85,B 0,C 180,E1 -21318.758,E2 -21318.758} C_VEL
LIN {X 0,Y 197.575,Z 699.645,A -85,B 0,C 180,E1 -21321.82,E2 -21321.82} C_VEL
LIN {X 0,Y 197.295,Z 701.149,A -85,B 0,C 180,E1 -21323.865,E2 -21323.865} C_VEL
LIN {X 0,Y 197.209,Z 702.244,A -85,B 0,C 180,E1 -21326.275,E2 -21326.275} C_VEL
LIN {X 0,Y 197.342,Z 702.966,A -85,B 0,C 180,E1 -21330,E2 -21330} C_VEL
LIN {X 0,Y 197.214,Z 702.082,A -85,B 0,C 180,E1 -21334.087,E2 -21334.087} C_VEL
LIN {X 0,Y 197.318,Z 701.149,A -85,B 0,C 180,E1 -21336.134,E2 -21336.134} C_VEL
LIN {X 0,Y 198.028,Z 697.796,A -85,B 0,C 180,E1 -21340.221,E2 -21340.221} C_VEL
LIN {X 0,Y 199.003,Z 694.164,A -85,B 0,C 180,E1 -21343.271,E2 -21343.271} C_VEL
LIN {X 0,Y 200.517,Z 689.431,A -85,B 0,C 180,E1 -21346.284,E2 -21346.284} C_VEL
LIN {X 0,Y 202.536,Z 683.458,A -85,B 0,C 180,E1 -21349.247,E2 -21349.247} C_VEL
LIN {X 0,Y 204.69,Z 677.369,A -85,B 0,C 180,E1 -21351.66,E2 -21351.66} C_VEL
LIN {X 0,Y 206.491,Z 671.599,A -85,B 0,C 180,E1 -21353.582,E2 -21353.582} C_VEL
LIN {X 0,Y 208.553,Z 664.969,A -85,B 0,C 180,E1 -21355.446,E2 -21355.446} C_VEL
LIN {X 0,Y 210.952,Z 657.146,A -85,B 0,C 180,E1 -21357.264,E2 -21357.264} C_VEL
LIN {X 0,Y 213.185,Z 649.065,A -85,B 0,C 180,E1 -21358.825,E2 -21358.825} C_VEL
LIN {X 0,Y 215.646,Z 639.308,A -85,B 0,C 180,E1 -21360.341,E2 -21360.341} C_VEL
LIN {X 0,Y 217.511,Z 630.923,A -85,B 0,C 180,E1 -21361.4,E2 -21361.4} C_VEL
LIN {X 0,Y 219.336,Z 620.417,A -85,B 0,C 180,E1 -21362.459,E2 -21362.459} C_VEL
LIN {X 0,Y 220.934,Z 609.937,A -85,B 0,C 180,E1 -21363.224,E2 -21363.224} C_VEL
LIN {X 0,Y 222.021,Z 599.974,A -85,B 0,C 180,E1 -21363.744,E2 -21363.744} C_VEL
LIN {X 0,Y 223.107,Z 578.226,A -85,B 0,C 180,E1 -21364.479,E2 -21364.479} C_VEL
LIN {X 0,Y 224.208,Z 551.576,A -85,B 0,C 180,E1 -21365.303,E2 -21365.303} C_VEL
LIN {X 0,Y 221.232,Z 533.274,A -85,B 0,C 180,E1 -21366.567,E2 -21366.567} C_VEL
LIN {X 0,Y 215.778,Z 520.106,A -85,B 0,C 180,E1 -21368.184,E2 -21368.184} C_VEL
LIN {X 0,Y 208.602,Z 505.297,A -85,B 0,C 180,E1 -21370.39,E2 -21370.39} C_VEL
LIN {X 0,Y 202.882,Z 495.321,A -85,B 0,C 180,E1 -21372.233,E2 -21372.233} C_VEL
LIN {X 0,Y 200.863,Z 491.456,A -85,B 0,C 180,E1 -21373.018,E2 -21373.018} C_VEL
LIN {X 0,Y 200.317,Z 489.109,A -85,B 0,C 180,E1 -21374.562,E2 -21374.562} C_VEL
LIN {X 0,Y 199.612,Z 486.171,A -85,B 0,C 180,E1 -21377.054,E2 -21377.054} C_VEL
LIN {X 0,Y 199.601,Z 486.104,A -85,B 0,C 180,E1 -21380.77,E2 -21380.77} C_VEL
LIN {X 0,Y 199.616,Z 486.106,A -85,B 0,C 180,E1 -21384.073,E2 -21384.073} C_VEL
LIN {X 0,Y 199.688,Z 486.096,A -85,B 0,C 180,E1 -21388.132,E2 -21388.132} C_VEL
LIN {X 0,Y 199.626,Z 486.081,A -85,B 0,C 180,E1 -21392.76,E2 -21392.76} C_VEL
LIN {X 0,Y 199.669,Z 486.111,A -85,B 0,C 180,E1 -21397.218,E2 -21397.218} C_VEL
LIN {X 0,Y 199.734,Z 486.058,A -85,B 0,C 180,E1 -21401.811,E2 -21401.811} C_VEL
LIN {X 0,Y 199.762,Z 486.098,A -85,B 0,C 180,E1 -21405.74,E2 -21405.74} C_VEL
LIN {X 0,Y 200.023,Z 486.02,A -85,B 0,C 180,E1 -21409.879,E2 -21409.879} C_VEL
LIN {X 0,Y 199.993,Z 486.06,A -85,B 0,C 180,E1 -21413.945,E2 -21413.945} C_VEL
LIN {X 0,Y 200.28,Z 486.009,A -85,B 0,C 180,E1 -21417.986,E2 -21417.986} C_VEL
LIN {X 0,Y 200.441,Z 485.966,A -85,B 0,C 180,E1 -21419.997,E2 -21419.997} C_VEL
LIN {X 0,Y 199.978,Z 486.067,A -85,B 0,C 180,E1 -21424.027,E2 -21424.027} C_VEL
LIN {X 0,Y 200.065,Z 486.03,A -85,B 0,C 180,E1 -21428.074,E2 -21428.074} C_VEL
LIN {X 0,Y 199.85,Z 486.057,A -85,B 0,C 180,E1 -21432.178,E2 -21432.178} C_VEL
LIN {X 0,Y 199.739,Z 486.091,A -85,B 0,C 180,E1 -21436.346,E2 -21436.346} C_VEL
LIN {X 0,Y 199.636,Z 486.08,A -85,B 0,C 180,E1 -21440.609,E2 -21440.609} C_VEL
LIN {X 0,Y 199.612,Z 486.107,A -85,B 0,C 180,E1 -21444.989,E2 -21444.989} C_VEL
LIN {X 0,Y 199.596,Z 486.102,A -85,B 0,C 180,E1 -21449.531,E2 -21449.531} C_VEL
LIN {X 0,Y 199.656,Z 486.106,A -85,B 0,C 180,E1 -21452.349,E2 -21452.349} C_VEL
LIN {X 0,Y 199.607,Z 486.11,A -85,B 0,C 180,E1 -21456.762,E2 -21456.762} C_VEL
LIN {X 0,Y 199.584,Z 486.109,A -85,B 0,C 180,E1 -21459.329,E2 -21459.329} C_VEL
LIN {X 0,Y 199.554,Z 486.114,A -85,B 0,C 180,E1 -21462.304,E2 -21462.304} C_VEL
LIN {X 0,Y 199.599,Z 486.319,A -85,B 0,C 180,E1 -21466.512,E2 -21466.512} C_VEL
LIN {X 0,Y 199.824,Z 487.298,A -85,B 0,C 180,E1 -21466.939,E2 -21466.939} C_VEL
LIN {X 0,Y 201.425,Z 490.072,A -85,B 0,C 180,E1 -21467.532,E2 -21467.532} C_VEL
LIN {X 0,Y 202.668,Z 491.489,A -85,B 0,C 180,E1 -21467.921,E2 -21467.921} C_VEL
LIN {X 0,Y 205.024,Z 495.001,A -85,B 0,C 180,E1 -21468.678,E2 -21468.678} C_VEL
LIN {X 0,Y 213.913,Z 509.261,A -85,B 0,C 180,E1 -21471.358,E2 -21471.358} C_VEL
LIN {X 0,Y 221.842,Z 524.131,A -85,B 0,C 180,E1 -21473.578,E2 -21473.578} C_VEL
LIN {X 0,Y 230.849,Z 542.476,A -85,B 0,C 180,E1 -21475.901,E2 -21475.901} C_VEL
LIN {X 0,Y 239.027,Z 555.508,A -85,B 0,C 180,E1 -21477.684,E2 -21477.684} C_VEL
LIN {X 0,Y 247.051,Z 566.251,A -85,B 0,C 180,E1 -21479.219,E2 -21479.219} C_VEL
LIN {X 0,Y 259.975,Z 580.795,A -85,B 0,C 180,E1 -21481.365,E2 -21481.365} C_VEL
LIN {X 0,Y 271.677,Z 592.222,A -85,B 0,C 180,E1 -21483.18,E2 -21483.18} C_VEL
LIN {X 0,Y 283.108,Z 602.248,A -85,B 0,C 180,E1 -21484.965,E2 -21484.965} C_VEL
LIN {X 0,Y 297.393,Z 613.62,A -85,B 0,C 180,E1 -21487.161,E2 -21487.161} C_VEL
LIN {X 0,Y 305.735,Z 619.985,A -85,B 0,C 180,E1 -21488.579,E2 -21488.579} C_VEL
LIN {X 0,Y 313.831,Z 625.862,A -85,B 0,C 180,E1 -21490.138,E2 -21490.138} C_VEL
LIN {X 0,Y 321.707,Z 631.42,A -85,B 0,C 180,E1 -21491.854,E2 -21491.854} C_VEL
LIN {X 0,Y 329.351,Z 636.879,A -85,B 0,C 180,E1 -21493.782,E2 -21493.782} C_VEL
LIN {X 0,Y 335.156,Z 640.718,A -85,B 0,C 180,E1 -21495.426,E2 -21495.426} C_VEL
LIN {X 0,Y 341.069,Z 644.309,A -85,B 0,C 180,E1 -21497.309,E2 -21497.309} C_VEL
LIN {X 0,Y 344.182,Z 646.628,A -85,B 0,C 180,E1 -21498.547,E2 -21498.547} C_VEL
LIN {X 0,Y 346.355,Z 648.174,A -85,B 0,C 180,E1 -21499.478,E2 -21499.478} C_VEL
LIN {X 0,Y 349.078,Z 649.891,A -85,B 0,C 180,E1 -21500.731,E2 -21500.731} C_VEL
LIN {X 0,Y 351.439,Z 651.257,A -85,B 0,C 180,E1 -21501.953,E2 -21501.953} C_VEL
LIN {X 0,Y 353.781,Z 652.482,A -85,B 0,C 180,E1 -21503.327,E2 -21503.327} C_VEL
LIN {X 0,Y 355.249,Z 653.138,A -85,B 0,C 180,E1 -21504.323,E2 -21504.323} C_VEL
LIN {X 0,Y 356.685,Z 653.723,A -85,B 0,C 180,E1 -21505.48,E2 -21505.48} C_VEL
LIN {X 0,Y 357.857,Z 654.034,A -85,B 0,C 180,E1 -21506.622,E2 -21506.622} C_VEL
LIN {X 0,Y 358.648,Z 654.477,A -85,B 0,C 180,E1 -21507.924,E2 -21507.924} C_VEL
LIN {X 0,Y 359.17,Z 654.613,A -85,B 0,C 180,E1 -21510,E2 -21510} C_VEL
LIN {X 0,Y 358.636,Z 654.483,A -85,B 0,C 180,E1 -21512.022,E2 -21512.022} C_VEL
LIN {X 0,Y 357.826,Z 654.031,A -85,B 0,C 180,E1 -21513.378,E2 -21513.378} C_VEL
LIN {X 0,Y 356.663,Z 653.7,A -85,B 0,C 180,E1 -21514.521,E2 -21514.521} C_VEL
LIN {X 0,Y 355.226,Z 653.117,A -85,B 0,C 180,E1 -21515.677,E2 -21515.677} C_VEL
LIN {X 0,Y 353.462,Z 652.319,A -85,B 0,C 180,E1 -21516.852,E2 -21516.852} C_VEL
LIN {X 0,Y 351.382,Z 651.292,A -85,B 0,C 180,E1 -21518.048,E2 -21518.048} C_VEL
LIN {X 0,Y 348.95,Z 649.873,A -85,B 0,C 180,E1 -21519.307,E2 -21519.307} C_VEL
LIN {X 0,Y 346.323,Z 648.178,A -85,B 0,C 180,E1 -21520.523,E2 -21520.523} C_VEL
LIN {X 0,Y 343.277,Z 645.987,A -85,B 0,C 180,E1 -21521.814,E2 -21521.814} C_VEL
LIN {X 0,Y 339.364,Z 643.274,A -85,B 0,C 180,E1 -21523.271,E2 -21523.271} C_VEL
LIN {X 0,Y 334.359,Z 640.247,A -85,B 0,C 180,E1 -21524.795,E2 -21524.795} C_VEL
LIN {X 0,Y 328.003,Z 635.864,A -85,B 0,C 180,E1 -21526.584,E2 -21526.584} C_VEL
LIN {X 0,Y 321.716,Z 631.416,A -85,B 0,C 180,E1 -21528.151,E2 -21528.151} C_VEL
LIN {X 0,Y 313.834,Z 625.865,A -85,B 0,C 180,E1 -21529.864,E2 -21529.864} C_VEL
LIN {X 0,Y 308.479,Z 621.884,A -85,B 0,C 180,E1 -21530.925,E2 -21530.925} C_VEL
LIN {X 0,Y 300.191,Z 615.832,A -85,B 0,C 180,E1 -21532.375,E2 -21532.375} C_VEL
LIN {X 0,Y 290.238,Z 608.146,A -85,B 0,C 180,E1 -21533.928,E2 -21533.928} C_VEL
LIN {X 0,Y 275.768,Z 596.017,A -85,B 0,C 180,E1 -21536.168,E2 -21536.168} C_VEL
LIN {X 0,Y 264.849,Z 585.705,A -85,B 0,C 180,E1 -21537.88,E2 -21537.88} C_VEL
LIN {X 0,Y 251.225,Z 571.256,A -85,B 0,C 180,E1 -21540.048,E2 -21540.048} C_VEL
LIN {X 0,Y 241.529,Z 559.096,A -85,B 0,C 180,E1 -21541.815,E2 -21541.815} C_VEL
LIN {X 0,Y 232.977,Z 546.147,A -85,B 0,C 180,E1 -21543.609,E2 -21543.609} C_VEL
LIN {X 0,Y 225.867,Z 532.716,A -85,B 0,C 180,E1 -21545.338,E2 -21545.338} C_VEL
LIN {X 0,Y 219.38,Z 519.324,A -85,B 0,C 180,E1 -21547.095,E2 -21547.095} C_VEL
LIN {X 0,Y 212.771,Z 507.443,A -85,B 0,C 180,E1 -21548.968,E2 -21548.968} C_VEL
LIN {X 0,Y 204.881,Z 494.841,A -85,B 0,C 180,E1 -21551.364,E2 -21551.364} C_VEL
LIN {X 0,Y 202.534,Z 491.233,A -85,B 0,C 180,E1 -21552.125,E2 -21552.125} C_VEL
LIN {X 0,Y 200.379,Z 488.557,A -85,B 0,C 180,E1 -21552.817,E2 -21552.817} C_VEL
LIN {X 0,Y 199.663,Z 486.652,A -85,B 0,C 180,E1 -21553.26,E2 -21553.26} C_VEL
LIN {X 0,Y 199.579,Z 486.202,A -85,B 0,C 180,E1 -21553.646,E2 -21553.646} C_VEL
LIN {X 0,Y 199.558,Z 486.11,A -85,B 0,C 180,E1 -21558.004,E2 -21558.004} C_VEL
LIN {X 0,Y 199.586,Z 486.109,A -85,B 0,C 180,E1 -21560.775,E2 -21560.775} C_VEL
LIN {X 0,Y 199.6,Z 486.094,A -85,B 0,C 180,E1 -21565.715,E2 -21565.715} C_VEL
LIN {X 0,Y 199.676,Z 486.111,A -85,B 0,C 180,E1 -21568.137,E2 -21568.137} C_VEL
LIN {X 0,Y 199.614,Z 486.084,A -85,B 0,C 180,E1 -21572.765,E2 -21572.765} C_VEL
LIN {X 0,Y 199.663,Z 486.11,A -85,B 0,C 180,E1 -21577.224,E2 -21577.224} C_VEL
LIN {X 0,Y 199.74,Z 486.064,A -85,B 0,C 180,E1 -21581.806,E2 -21581.806} C_VEL
LIN {X 0,Y 199.79,Z 486.097,A -85,B 0,C 180,E1 -21585.748,E2 -21585.748} C_VEL
LIN {X 0,Y 200.019,Z 486.02,A -85,B 0,C 180,E1 -21589.885,E2 -21589.885} C_VEL
LIN {X 0,Y 199.993,Z 486.07,A -85,B 0,C 180,E1 -21593.952,E2 -21593.952} C_VEL
LIN {X 0,Y 200.267,Z 485.996,A -85,B 0,C 180,E1 -21597.992,E2 -21597.992} C_VEL
LIN {X 0,Y 200.441,Z 485.966,A -85,B 0,C 180,E1 -21600.003,E2 -21600.003} C_VEL
LIN {X 0,Y 199.979,Z 486.074,A -85,B 0,C 180,E1 -21604.034,E2 -21604.034} C_VEL
LIN {X 0,Y 200.064,Z 486.018,A -85,B 0,C 180,E1 -21608.081,E2 -21608.081} C_VEL
LIN {X 0,Y 200.005,Z 486.023,A -85,B 0,C 180,E1 -21610.3,E2 -21610.3} C_VEL
LIN {X 0,Y 199.736,Z 486.073,A -85,B 0,C 180,E1 -21616.352,E2 -21616.352} C_VEL
LIN {X 0,Y 199.641,Z 486.088,A -85,B 0,C 180,E1 -21620.615,E2 -21620.615} C_VEL
LIN {X 0,Y 199.622,Z 486.09,A -85,B 0,C 180,E1 -21624.994,E2 -21624.994} C_VEL
LIN {X 0,Y 199.607,Z 486.113,A -85,B 0,C 180,E1 -21629.536,E2 -21629.536} C_VEL
LIN {X 0,Y 199.667,Z 486.092,A -85,B 0,C 180,E1 -21632.354,E2 -21632.354} C_VEL
LIN {X 0,Y 199.621,Z 486.119,A -85,B 0,C 180,E1 -21636.767,E2 -21636.767} C_VEL
LIN {X 0,Y 199.599,Z 486.104,A -85,B 0,C 180,E1 -21639.334,E2 -21639.334} C_VEL
LIN {X 0,Y 199.625,Z 486.238,A -85,B 0,C 180,E1 -21643.105,E2 -21643.105} C_VEL
LIN {X 0,Y 200.711,Z 490.881,A -85,B 0,C 180,E1 -21646.72,E2 -21646.72} C_VEL
LIN {X 0,Y 201.128,Z 492.175,A -85,B 0,C 180,E1 -21647.132,E2 -21647.132} C_VEL
LIN {X 0,Y 203.513,Z 496.146,A -85,B 0,C 180,E1 -21647.965,E2 -21647.965} C_VEL
LIN {X 0,Y 209.95,Z 508.017,A -85,B 0,C 180,E1 -21650.039,E2 -21650.039} C_VEL
LIN {X 0,Y 216.885,Z 522.601,A -85,B 0,C 180,E1 -21652.147,E2 -21652.147} C_VEL
LIN {X 0,Y 221.509,Z 534.323,A -85,B 0,C 180,E1 -21653.527,E2 -21653.527} C_VEL
LIN {X 0,Y 224.285,Z 552.503,A -85,B 0,C 180,E1 -21654.746,E2 -21654.746} C_VEL
LIN {X 0,Y 222.144,Z 597.895,A -85,B 0,C 180,E1 -21656.165,E2 -21656.165} C_VEL
LIN {X 0,Y 221.197,Z 607.857,A -85,B 0,C 180,E1 -21656.657,E2 -21656.657} C_VEL
LIN {X 0,Y 219.984,Z 616.632,A -85,B 0,C 180,E1 -21657.241,E2 -21657.241} C_VEL
LIN {X 0,Y 218.643,Z 625.019,A -85,B 0,C 180,E1 -21657.97,E2 -21657.97} C_VEL
LIN {X 0,Y 216.332,Z 636.128,A -85,B 0,C 180,E1 -21659.225,E2 -21659.225} C_VEL
LIN {X 0,Y 214.229,Z 645.128,A -85,B 0,C 180,E1 -21660.522,E2 -21660.522} C_VEL
LIN {X 0,Y 211.852,Z 653.851,A -85,B 0,C 180,E1 -21662.058,E2 -21662.058} C_VEL
LIN {X 0,Y 210.857,Z 657.474,A -85,B 0,C 180,E1 -21662.803,E2 -21662.803} C_VEL
LIN {X 0,Y 208.937,Z 661.962,A -85,B 0,C 180,E1 -21663.714,E2 -21663.714} C_VEL
LIN {X 0,Y 204.157,Z 668.803,A -85,B 0,C 180,E1 -21665.197,E2 -21665.197} C_VEL
LIN {X 0,Y 199.411,Z 675.186,A -85,B 0,C 180,E1 -21666.9,E2 -21666.9} C_VEL
LIN {X 0,Y 197.571,Z 678.662,A -85,B 0,C 180,E1 -21668.143,E2 -21668.143} C_VEL
LIN {X 0,Y 195.468,Z 684.355,A -85,B 0,C 180,E1 -21670.575,E2 -21670.575} C_VEL
LIN {X 0,Y 193.674,Z 689.233,A -85,B 0,C 180,E1 -21673.124,E2 -21673.124} C_VEL
LIN {X 0,Y 192.051,Z 693.967,A -85,B 0,C 180,E1 -21676.24,E2 -21676.24} C_VEL
LIN {X 0,Y 191.016,Z 697.599,A -85,B 0,C 180,E1 -21679.399,E2 -21679.399} C_VEL
LIN {X 0,Y 190.222,Z 700.952,A -85,B 0,C 180,E1 -21683.636,E2 -21683.636} C_VEL
LIN {X 0,Y 190.108,Z 702.225,A -85,B 0,C 180,E1 -21686.553,E2 -21686.553} C_VEL
LIN {X 0,Y 190.246,Z 702.77,A -85,B 0,C 180,E1 -21690,E2 -21690} C_VEL
LIN {X 0,Y 190.136,Z 701.886,A -85,B 0,C 180,E1 -21694.239,E2 -21694.239} C_VEL
LIN {X 0,Y 190.238,Z 700.952,A -85,B 0,C 180,E1 -21696.363,E2 -21696.363} C_VEL
LIN {X 0,Y 191.016,Z 697.599,A -85,B 0,C 180,E1 -21700.601,E2 -21700.601} C_VEL
LIN {X 0,Y 192.051,Z 693.967,A -85,B 0,C 180,E1 -21703.76,E2 -21703.76} C_VEL
LIN {X 0,Y 193.674,Z 689.233,A -85,B 0,C 180,E1 -21706.876,E2 -21706.876} C_VEL
LIN {X 0,Y 195.812,Z 683.261,A -85,B 0,C 180,E1 -21709.936,E2 -21709.936} C_VEL
LIN {X 0,Y 198.069,Z 677.172,A -85,B 0,C 180,E1 -21712.422,E2 -21712.422} C_VEL
LIN {X 0,Y 200.463,Z 669.867,A -85,B 0,C 180,E1 -21714.879,E2 -21714.879} C_VEL
LIN {X 0,Y 203.346,Z 661.073,A -85,B 0,C 180,E1 -21717.254,E2 -21717.254} C_VEL
LIN {X 0,Y 206.641,Z 650.181,A -85,B 0,C 180,E1 -21719.548,E2 -21719.548} C_VEL
LIN {X 0,Y 209.201,Z 640.702,A -85,B 0,C 180,E1 -21721.098,E2 -21721.098} C_VEL
LIN {X 0,Y 211.472,Z 630.726,A -85,B 0,C 180,E1 -21722.404,E2 -21722.404} C_VEL
LIN {X 0,Y 213.392,Z 620.221,A -85,B 0,C 180,E1 -21723.48,E2 -21723.48} C_VEL
LIN {X 0,Y 215.017,Z 609.937,A -85,B 0,C 180,E1 -21724.246,E2 -21724.246} C_VEL
LIN {X 0,Y 216.185,Z 599.491,A -85,B 0,C 180,E1 -21724.799,E2 -21724.799} C_VEL
LIN {X 0,Y 217.364,Z 576.399,A -85,B 0,C 180,E1 -21725.59,E2 -21725.59} C_VEL
LIN {X 0,Y 218.349,Z 552.266,A -85,B 0,C 180,E1 -21726.364,E2 -21726.364} C_VEL
LIN {X 0,Y 215.777,Z 536.013,A -85,B 0,C 180,E1 -21727.529,E2 -21727.529} C_VEL
LIN {X 0,Y 210.364,Z 522.951,A -85,B 0,C 180,E1 -21729.222,E2 -21729.222} C_VEL
LIN {X 0,Y 203.972,Z 509.591,A -85,B 0,C 180,E1 -21731.301,E2 -21731.301} C_VEL
LIN {X 0,Y 198.326,Z 499.64,A -85,B 0,C 180,E1 -21733.222,E2 -21733.222} C_VEL
LIN {X 0,Y 195.522,Z 494.905,A -85,B 0,C 180,E1 -21734.23,E2 -21734.23} C_VEL
LIN {X 0,Y 193.56,Z 491.076,A -85,B 0,C 180,E1 -21735.105,E2 -21735.105} C_VEL
LIN {X 0,Y 192.539,Z 487.156,A -85,B 0,C 180,E1 -21738.211,E2 -21738.211} C_VEL
LIN {X 0,Y 192.586,Z 486.992,A -85,B 0,C 180,E1 -21743.401,E2 -21743.401} C_VEL
LIN {X 0,Y 192.608,Z 486.966,A -85,B 0,C 180,E1 -21747.059,E2 -21747.059} C_VEL
LIN {X 0,Y 192.614,Z 486.963,A -85,B 0,C 180,E1 -21751.681,E2 -21751.681} C_VEL
LIN {X 0,Y 192.657,Z 486.978,A -85,B 0,C 180,E1 -21756.339,E2 -21756.339} C_VEL
LIN {X 0,Y 192.687,Z 486.934,A -85,B 0,C 180,E1 -21761.496,E2 -21761.496} C_VEL
LIN {X 0,Y 192.697,Z 486.974,A -85,B 0,C 180,E1 -21765.205,E2 -21765.205} C_VEL
LIN {X 0,Y 192.946,Z 486.902,A -85,B 0,C 180,E1 -21769.564,E2 -21769.564} C_VEL
LIN {X 0,Y 192.958,Z 486.93,A -85,B 0,C 180,E1 -21773.724,E2 -21773.724} C_VEL
LIN {X 0,Y 193.224,Z 486.887,A -85,B 0,C 180,E1 -21777.912,E2 -21777.912} C_VEL
LIN {X 0,Y 193.408,Z 486.841,A -85,B 0,C 180,E1 -21779.997,E2 -21779.997} C_VEL
LIN {X 0,Y 192.926,Z 486.946,A -85,B 0,C 180,E1 -21784.175,E2 -21784.175} C_VEL
LIN {X 0,Y 193.017,Z 486.903,A -85,B 0,C 180,E1 -21788.371,E2 -21788.371} C_VEL
LIN {X 0,Y 192.776,Z 486.944,A -85,B 0,C 180,E1 -21792.632,E2 -21792.632} C_VEL
LIN {X 0,Y 192.681,Z 486.958,A -85,B 0,C 180,E1 -21796.962,E2 -21796.962} C_VEL
LIN {X 0,Y 192.57,Z 486.969,A -85,B 0,C 180,E1 -21801.401,E2 -21801.401} C_VEL
LIN {X 0,Y 192.611,Z 486.99,A -85,B 0,C 180,E1 -21804.19,E2 -21804.19} C_VEL
LIN {X 0,Y 192.587,Z 486.966,A -85,B 0,C 180,E1 -21808.859,E2 -21808.859} C_VEL
LIN {X 0,Y 192.585,Z 486.974,A -85,B 0,C 180,E1 -21813.184,E2 -21813.184} C_VEL
LIN {X 0,Y 192.531,Z 487,A -85,B 0,C 180,E1 -21818.352,E2 -21818.352} C_VEL
LIN {X 0,Y 192.495,Z 487.004,A -85,B 0,C 180,E1 -21823.097,E2 -21823.097} C_VEL
LIN {X 0,Y 192.57,Z 487.284,A -85,B 0,C 180,E1 -21824.64,E2 -21824.64} C_VEL
LIN {X 0,Y 192.891,Z 488.451,A -85,B 0,C 180,E1 -21825.046,E2 -21825.046} C_VEL
LIN {X 0,Y 194.499,Z 491.089,A -85,B 0,C 180,E1 -21825.674,E2 -21825.674} C_VEL
LIN {X 0,Y 195.701,Z 492.329,A -85,B 0,C 180,E1 -21826.081,E2 -21826.081} C_VEL
LIN {X 0,Y 197.813,Z 495.665,A -85,B 0,C 180,E1 -21826.834,E2 -21826.834} C_VEL
LIN {X 0,Y 203.719,Z 504.599,A -85,B 0,C 180,E1 -21828.796,E2 -21828.796} C_VEL
LIN {X 0,Y 210.536,Z 515.908,A -85,B 0,C 180,E1 -21830.902,E2 -21830.902} C_VEL
LIN {X 0,Y 218.485,Z 531.482,A -85,B 0,C 180,E1 -21833.218,E2 -21833.218} C_VEL
LIN {X 0,Y 225.482,Z 545.951,A -85,B 0,C 180,E1 -21835.098,E2 -21835.098} C_VEL
LIN {X 0,Y 233.829,Z 559.581,A -85,B 0,C 180,E1 -21837.015,E2 -21837.015} C_VEL
LIN {X 0,Y 242.57,Z 571.391,A -85,B 0,C 180,E1 -21838.757,E2 -21838.757} C_VEL
LIN {X 0,Y 255.188,Z 585.757,A -85,B 0,C 180,E1 -21840.969,E2 -21840.969} C_VEL
LIN {X 0,Y 265.931,Z 596.535,A -85,B 0,C 180,E1 -21842.799,E2 -21842.799} C_VEL
LIN {X 0,Y 276.265,Z 605.83,A -85,B 0,C 180,E1 -21844.559,E2 -21844.559} C_VEL
LIN {X 0,Y 290.358,Z 617.086,A -85,B 0,C 180,E1 -21846.886,E2 -21846.886} C_VEL
LIN {X 0,Y 300.165,Z 624.621,A -85,B 0,C 180,E1 -21848.536,E2 -21848.536} C_VEL
LIN {X 0,Y 307.952,Z 630.248,A -85,B 0,C 180,E1 -21849.982,E2 -21849.982} C_VEL
LIN {X 0,Y 314.989,Z 635.381,A -85,B 0,C 180,E1 -21851.481,E2 -21851.481} C_VEL
LIN {X 0,Y 322.052,Z 640.309,A -85,B 0,C 180,E1 -21853.167,E2 -21853.167} C_VEL
LIN {X 0,Y 327.816,Z 644.317,A -85,B 0,C 180,E1 -21854.732,E2 -21854.732} C_VEL
LIN {X 0,Y 334.126,Z 648.254,A -85,B 0,C 180,E1 -21856.622,E2 -21856.622} C_VEL
LIN {X 0,Y 338.021,Z 650.877,A -85,B 0,C 180,E1 -21858,E2 -21858} C_VEL
LIN {X 0,Y 342.592,Z 654.1,A -85,B 0,C 180,E1 -21859.944,E2 -21859.944} C_VEL
LIN {X 0,Y 347.424,Z 656.954,A -85,B 0,C 180,E1 -21862.381,E2 -21862.381} C_VEL
LIN {X 0,Y 350.379,Z 658.394,A -85,B 0,C 180,E1 -21864.244,E2 -21864.244} C_VEL
LIN {X 0,Y 352.32,Z 659.16,A -85,B 0,C 180,E1 -21865.823,E2 -21865.823} C_VEL
LIN {X 0,Y 353.128,Z 659.371,A -85,B 0,C 180,E1 -21866.577,E2 -21866.577} C_VEL
LIN {X 0,Y 353.863,Z 659.769,A -85,B 0,C 180,E1 -21867.724,E2 -21867.724} C_VEL
LIN {X 0,Y 354.257,Z 660.041,A -85,B 0,C 180,E1 -21868.863,E2 -21868.863} C_VEL
LIN {X 0,Y 354.536,Z 659.967,A -85,B 0,C 180,E1 -21870,E2 -21870} C_VEL
LIN {X 0,Y 354.277,Z 660.003,A -85,B 0,C 180,E1 -21871.137,E2 -21871.137} C_VEL
LIN {X 0,Y 353.837,Z 659.766,A -85,B 0,C 180,E1 -21872.277,E2 -21872.277} C_VEL
LIN {X 0,Y 352.33,Z 659.157,A -85,B 0,C 180,E1 -21874.199,E2 -21874.199} C_VEL
LIN {X 0,Y 350.363,Z 658.361,A -85,B 0,C 180,E1 -21875.756,E2 -21875.756} C_VEL
LIN {X 0,Y 347.422,Z 657.011,A -85,B 0,C 180,E1 -21877.617,E2 -21877.617} C_VEL
LIN {X 0,Y 342.586,Z 654.126,A -85,B 0,C 180,E1 -21880.051,E2 -21880.051} C_VEL
LIN {X 0,Y 337.993,Z 650.842,A -85,B 0,C 180,E1 -21882.001,E2 -21882.001} C_VEL
LIN {X 0,Y 334.145,Z 648.266,A -85,B 0,C 180,E1 -21883.377,E2 -21883.377} C_VEL
LIN {X 0,Y 327.813,Z 644.322,A -85,B 0,C 180,E1 -21885.267,E2 -21885.267} C_VEL
LIN {X 0,Y 322.761,Z 640.766,A -85,B 0,C 180,E1 -21886.657,E2 -21886.657} C_VEL
LIN {X 0,Y 316.938,Z 636.658,A -85,B 0,C 180,E1 -21888.086,E2 -21888.086} C_VEL
LIN {X 0,Y 309.691,Z 631.557,A -85,B 0,C 180,E1 -21889.657,E2 -21889.657} C_VEL
LIN {X 0,Y 301.56,Z 625.614,A -85,B 0,C 180,E1 -21891.224,E2 -21891.224} C_VEL
LIN {X 0,Y 292.347,Z 618.59,A -85,B 0,C 180,E1 -21892.796,E2 -21892.796} C_VEL
LIN {X 0,Y 279.091,Z 608.129,A -85,B 0,C 180,E1 -21894.975,E2 -21894.975} C_VEL
LIN {X 0,Y 268.929,Z 599.258,A -85,B 0,C 180,E1 -21896.699,E2 -21896.699} C_VEL
LIN {X 0,Y 259.45,Z 590.076,A -85,B 0,C 180,E1 -21898.32,E2 -21898.32} C_VEL
LIN {X 0,Y 248.826,Z 578.772,A -85,B 0,C 180,E1 -21900.125,E2 -21900.125} C_VEL
LIN {X 0,Y 237.482,Z 564.825,A -85,B 0,C 180,E1 -21902.227,E2 -21902.227} C_VEL
LIN {X 0,Y 228.365,Z 551.016,A -85,B 0,C 180,E1 -21904.206,E2 -21904.206} C_VEL
LIN {X 0,Y 221.217,Z 537.518,A -85,B 0,C 180,E1 -21906.013,E2 -21906.013} C_VEL
LIN {X 0,Y 214.347,Z 523.115,A -85,B 0,C 180,E1 -21907.968,E2 -21907.968} C_VEL
LIN {X 0,Y 207.502,Z 510.664,A -85,B 0,C 180,E1 -21910.02,E2 -21910.02} C_VEL
LIN {X 0,Y 200.293,Z 499.318,A -85,B 0,C 180,E1 -21912.325,E2 -21912.325} C_VEL
LIN {X 0,Y 197.667,Z 495.509,A -85,B 0,C 180,E1 -21913.213,E2 -21913.213} C_VEL
LIN {X 0,Y 195.059,Z 491.607,A -85,B 0,C 180,E1 -21914.139,E2 -21914.139} C_VEL
LIN {X 0,Y 193.212,Z 489.244,A -85,B 0,C 180,E1 -21914.798,E2 -21914.798} C_VEL
LIN {X 0,Y 192.61,Z 487.478,A -85,B 0,C 180,E1 -21915.246,E2 -21915.246} C_VEL
LIN {X 0,Y 192.492,Z 487.033,A -85,B 0,C 180,E1 -21915.834,E2 -21915.834} C_VEL
LIN {X 0,Y 192.494,Z 486.986,A -85,B 0,C 180,E1 -21920.059,E2 -21920.059} C_VEL
LIN {X 0,Y 192.548,Z 486.976,A -85,B 0,C 180,E1 -21924.272,E2 -21924.272} C_VEL
LIN {X 0,Y 192.596,Z 486.976,A -85,B 0,C 180,E1 -21927.064,E2 -21927.064} C_VEL
LIN {X 0,Y 192.603,Z 486.959,A -85,B 0,C 180,E1 -21931.686,E2 -21931.686} C_VEL
LIN {X 0,Y 192.65,Z 486.989,A -85,B 0,C 180,E1 -21936.345,E2 -21936.345} C_VEL
LIN {X 0,Y 192.689,Z 486.94,A -85,B 0,C 180,E1 -21941.495,E2 -21941.495} C_VEL
LIN {X 0,Y 192.717,Z 486.98,A -85,B 0,C 180,E1 -21945.214,E2 -21945.214} C_VEL
LIN {X 0,Y 192.942,Z 486.901,A -85,B 0,C 180,E1 -21949.57,E2 -21949.57} C_VEL
LIN {X 0,Y 192.957,Z 486.945,A -85,B 0,C 180,E1 -21953.73,E2 -21953.73} C_VEL
LIN {X 0,Y 193.213,Z 486.874,A -85,B 0,C 180,E1 -21957.919,E2 -21957.919} C_VEL
LIN {X 0,Y 193.408,Z 486.841,A -85,B 0,C 180,E1 -21960.003,E2 -21960.003} C_VEL
LIN {X 0,Y 192.927,Z 486.954,A -85,B 0,C 180,E1 -21964.181,E2 -21964.181} C_VEL
LIN {X 0,Y 193.017,Z 486.892,A -85,B 0,C 180,E1 -21968.378,E2 -21968.378} C_VEL
LIN {X 0,Y 192.752,Z 486.961,A -85,B 0,C 180,E1 -21972.64,E2 -21972.64} C_VEL
LIN {X 0,Y 192.677,Z 486.943,A -85,B 0,C 180,E1 -21976.969,E2 -21976.969} C_VEL
LIN {X 0,Y 192.575,Z 486.981,A -85,B 0,C 180,E1 -21981.408,E2 -21981.408} C_VEL
LIN {X 0,Y 192.619,Z 486.973,A -85,B 0,C 180,E1 -21984.196,E2 -21984.196} C_VEL
LIN {X 0,Y 192.597,Z 486.973,A -85,B 0,C 180,E1 -21988.864,E2 -21988.864} C_VEL
LIN {X 0,Y 192.597,Z 486.965,A -85,B 0,C 180,E1 -21993.189,E2 -21993.189} C_VEL
LIN {X 0,Y 192.546,Z 486.988,A -85,B 0,C 180,E1 -21998.357,E2 -21998.357} C_VEL
LIN {X 0,Y 192.559,Z 487.134,A -85,B 0,C 180,E1 -22001.782,E2 -22001.782} C_VEL
LIN {X 0,Y 193.578,Z 491.044,A -85,B 0,C 180,E1 -22004.889,E2 -22004.889} C_VEL
LIN {X 0,Y 195.672,Z 495.122,A -85,B 0,C 180,E1 -22005.823,E2 -22005.823} C_VEL
LIN {X 0,Y 200.441,Z 503.344,A -85,B 0,C 180,E1 -22007.516,E2 -22007.516} C_VEL
LIN {X 0,Y 205.379,Z 512.396,A -85,B 0,C 180,E1 -22009.167,E2 -22009.167} C_VEL
LIN {X 0,Y 212.115,Z 526.9,A -85,B 0,C 180,E1 -22011.328,E2 -22011.328} C_VEL
LIN {X 0,Y 216.025,Z 537.001,A -85,B 0,C 180,E1 -22012.562,E2 -22012.562} C_VEL
LIN {X 0,Y 218.472,Z 552.966,A -85,B 0,C 180,E1 -22013.687,E2 -22013.687} C_VEL
LIN {X 0,Y 216.285,Z 597.446,A -85,B 0,C 180,E1 -22015.104,E2 -22015.104} C_VEL
LIN {X 0,Y 215.279,Z 607.905,A -85,B 0,C 180,E1 -22015.634,E2 -22015.634} C_VEL
LIN {X 0,Y 213.847,Z 617.698,A -85,B 0,C 180,E1 -22016.318,E2 -22016.318} C_VEL
LIN {X 0,Y 212.276,Z 626.791,A -85,B 0,C 180,E1 -22017.171,E2 -22017.171} C_VEL
LIN {X 0,Y 210.251,Z 635.932,A -85,B 0,C 180,E1 -22018.233,E2 -22018.233} C_VEL
LIN {X 0,Y 208.06,Z 644.931,A -85,B 0,C 180,E1 -22019.557,E2 -22019.557} C_VEL
LIN {X 0,Y 205.6,Z 653.654,A -85,B 0,C 180,E1 -22021.13,E2 -22021.13} C_VEL
LIN {X 0,Y 203.36,Z 661.073,A -85,B 0,C 180,E1 -22022.748,E2 -22022.748} C_VEL
LIN {X 0,Y 200.445,Z 669.866,A -85,B 0,C 180,E1 -22025.119,E2 -22025.119} C_VEL
LIN {X 0,Y 198.29,Z 676.569,A -85,B 0,C 180,E1 -22027.351,E2 -22027.351} C_VEL
LIN {X 0,Y 197.571,Z 678.662,A -85,B 0,C 180,E1 -22028.143,E2 -22028.143} C_VEL
LIN {X 0,Y 195.741,Z 682.086,A -85,B 0,C 180,E1 -22029.451,E2 -22029.451} C_VEL
LIN {X 0,Y 191.073,Z 687.042,A -85,B 0,C 180,E1 -22031.594,E2 -22031.594} C_VEL
LIN {X 0,Y 186.625,Z 691.377,A -85,B 0,C 180,E1 -22033.956,E2 -22033.956} C_VEL
LIN {X 0,Y 185.181,Z 693.582,A -85,B 0,C 180,E1 -22035.572,E2 -22035.572} C_VEL
LIN {X 0,Y 184.324,Z 696.31,A -85,B 0,C 180,E1 -22037.895,E2 -22037.895} C_VEL
LIN {X 0,Y 183.502,Z 699.251,A -85,B 0,C 180,E1 -22041.188,E2 -22041.188} C_VEL
LIN {X 0,Y 183.145,Z 700.755,A -85,B 0,C 180,E1 -22043.389,E2 -22043.389} C_VEL
LIN {X 0,Y 183.02,Z 702.144,A -85,B 0,C 180,E1 -22046.808,E2 -22046.808} C_VEL
LIN {X 0,Y 183.153,Z 702.573,A -85,B 0,C 180,E1 -22050,E2 -22050} C_VEL
LIN {X 0,Y 183.04,Z 702.118,A -85,B 0,C 180,E1 -22053.301,E2 -22053.301} C_VEL
LIN {X 0,Y 183.185,Z 700.756,A -85,B 0,C 180,E1 -22056.609,E2 -22056.609} C_VEL
LIN {X 0,Y 183.995,Z 697.401,A -85,B 0,C 180,E1 -22061.01,E2 -22061.01} C_VEL
LIN {X 0,Y 185.124,Z 693.77,A -85,B 0,C 180,E1 -22064.286,E2 -22064.286} C_VEL
LIN {X 0,Y 186.861,Z 689.036,A -85,B 0,C 180,E1 -22067.511,E2 -22067.511} C_VEL
LIN {X 0,Y 189.134,Z 683.064,A -85,B 0,C 180,E1 -22070.671,E2 -22070.671} C_VEL
LIN {X 0,Y 190.917,Z 678.573,A -85,B 0,C 180,E1 -22072.614,E2 -22072.614} C_VEL
LIN {X 0,Y 192.864,Z 673.105,A -85,B 0,C 180,E1 -22074.66,E2 -22074.66} C_VEL
LIN {X 0,Y 195.789,Z 664.576,A -85,B 0,C 180,E1 -22077.237,E2 -22077.237} C_VEL
LIN {X 0,Y 198.376,Z 656.752,A -85,B 0,C 180,E1 -22079.152,E2 -22079.152} C_VEL
LIN {X 0,Y 200.863,Z 648.672,A -85,B 0,C 180,E1 -22080.778,E2 -22080.778} C_VEL
LIN {X 0,Y 203.503,Z 638.916,A -85,B 0,C 180,E1 -22082.364,E2 -22082.364} C_VEL
LIN {X 0,Y 205.494,Z 630.529,A -85,B 0,C 180,E1 -22083.468,E2 -22083.468} C_VEL
LIN {X 0,Y 207.518,Z 620.025,A -85,B 0,C 180,E1 -22084.56,E2 -22084.56} C_VEL
LIN {X 0,Y 209.151,Z 609.94,A -85,B 0,C 180,E1 -22085.33,E2 -22085.33} C_VEL
LIN {X 0,Y 210.422,Z 599.095,A -85,B 0,C 180,E1 -22085.908,E2 -22085.908} C_VEL
LIN {X 0,Y 211.634,Z 576.203,A -85,B 0,C 180,E1 -22086.708,E2 -22086.708} C_VEL
LIN {X 0,Y 212.634,Z 553.358,A -85,B 0,C 180,E1 -22087.453,E2 -22087.453} C_VEL
LIN {X 0,Y 210.173,Z 538.147,A -85,B 0,C 180,E1 -22088.612,E2 -22088.612} C_VEL
LIN {X 0,Y 204.489,Z 524.57,A -85,B 0,C 180,E1 -22090.496,E2 -22090.496} C_VEL
LIN {X 0,Y 198.977,Z 513.139,A -85,B 0,C 180,E1 -22092.399,E2 -22092.399} C_VEL
LIN {X 0,Y 191.98,Z 500.557,A -85,B 0,C 180,E1 -22094.969,E2 -22094.969} C_VEL
LIN {X 0,Y 188.791,Z 495.279,A -85,B 0,C 180,E1 -22096.22,E2 -22096.22} C_VEL
LIN {X 0,Y 186.399,Z 491.308,A -85,B 0,C 180,E1 -22097.256,E2 -22097.256} C_VEL
LIN {X 0,Y 186.033,Z 490.214,A -85,B 0,C 180,E1 -22097.775,E2 -22097.775} C_VEL
LIN {X 0,Y 185.474,Z 487.947,A -85,B 0,C 180,E1 -22099.893,E2 -22099.893} C_VEL
LIN {X 0,Y 185.505,Z 487.878,A -85,B 0,C 180,E1 -22102.711,E2 -22102.711} C_VEL
LIN {X 0,Y 185.533,Z 487.855,A -85,B 0,C 180,E1 -22107.969,E2 -22107.969} C_VEL
LIN {X 0,Y 185.493,Z 487.839,A -85,B 0,C 180,E1 -22112.954,E2 -22112.954} C_VEL
LIN {X 0,Y 185.545,Z 487.869,A -85,B 0,C 180,E1 -22117.739,E2 -22117.739} C_VEL
LIN {X 0,Y 185.63,Z 487.815,A -85,B 0,C 180,E1 -22122.366,E2 -22122.366} C_VEL
LIN {X 0,Y 185.683,Z 487.847,A -85,B 0,C 180,E1 -22126.871,E2 -22126.871} C_VEL
LIN {X 0,Y 185.968,Z 487.768,A -85,B 0,C 180,E1 -22131.302,E2 -22131.302} C_VEL
LIN {X 0,Y 186.17,Z 487.765,A -85,B 0,C 180,E1 -22137.833,E2 -22137.833} C_VEL
LIN {X 0,Y 186.373,Z 487.716,A -85,B 0,C 180,E1 -22139.997,E2 -22139.997} C_VEL
LIN {X 0,Y 185.874,Z 487.825,A -85,B 0,C 180,E1 -22144.334,E2 -22144.334} C_VEL
LIN {X 0,Y 185.968,Z 487.776,A -85,B 0,C 180,E1 -22148.691,E2 -22148.691} C_VEL
LIN {X 0,Y 185.702,Z 487.833,A -85,B 0,C 180,E1 -22153.121,E2 -22153.121} C_VEL
LIN {X 0,Y 185.619,Z 487.818,A -85,B 0,C 180,E1 -22158.818,E2 -22158.818} C_VEL
LIN {X 0,Y 185.538,Z 487.864,A -85,B 0,C 180,E1 -22164.62,E2 -22164.62} C_VEL
LIN {X 0,Y 185.509,Z 487.854,A -85,B 0,C 180,E1 -22169.501,E2 -22169.501} C_VEL
LIN {X 0,Y 185.519,Z 487.85,A -85,B 0,C 180,E1 -22173.549,E2 -22173.549} C_VEL
LIN {X 0,Y 185.49,Z 487.876,A -85,B 0,C 180,E1 -22177.312,E2 -22177.312} C_VEL
LIN {X 0,Y 185.435,Z 487.983,A -85,B 0,C 180,E1 -22182.227,E2 -22182.227} C_VEL
LIN {X 0,Y 185.685,Z 489.03,A -85,B 0,C 180,E1 -22182.782,E2 -22182.782} C_VEL
LIN {X 0,Y 187.297,Z 491.844,A -85,B 0,C 180,E1 -22183.506,E2 -22183.506} C_VEL
LIN {X 0,Y 188.834,Z 493.377,A -85,B 0,C 180,E1 -22184.081,E2 -22184.081} C_VEL
LIN {X 0,Y 190.886,Z 496.633,A -85,B 0,C 180,E1 -22184.888,E2 -22184.888} C_VEL
LIN {X 0,Y 192.487,Z 498.86,A -85,B 0,C 180,E1 -22185.483,E2 -22185.483} C_VEL
LIN {X 0,Y 197.984,Z 507.074,A -85,B 0,C 180,E1 -22187.436,E2 -22187.436} C_VEL
LIN {X 0,Y 205.505,Z 519.526,A -85,B 0,C 180,E1 -22189.907,E2 -22189.907} C_VEL
LIN {X 0,Y 212.638,Z 533.575,A -85,B 0,C 180,E1 -22192.11,E2 -22192.11} C_VEL
LIN {X 0,Y 220.966,Z 550.953,A -85,B 0,C 180,E1 -22194.468,E2 -22194.468} C_VEL
LIN {X 0,Y 229.46,Z 564.819,A -85,B 0,C 180,E1 -22196.492,E2 -22196.492} C_VEL
LIN {X 0,Y 237.993,Z 576.394,A -85,B 0,C 180,E1 -22198.255,E2 -22198.255} C_VEL
LIN {X 0,Y 249.346,Z 589.582,A -85,B 0,C 180,E1 -22200.377,E2 -22200.377} C_VEL
LIN {X 0,Y 261.381,Z 601.916,A -85,B 0,C 180,E1 -22202.645,E2 -22202.645} C_VEL
LIN {X 0,Y 273.58,Z 612.768,A -85,B 0,C 180,E1 -22204.889,E2 -22204.889} C_VEL
LIN {X 0,Y 287.48,Z 623.711,A -85,B 0,C 180,E1 -22207.342,E2 -22207.342} C_VEL
LIN {X 0,Y 298.67,Z 632.082,A -85,B 0,C 180,E1 -22209.332,E2 -22209.332} C_VEL
LIN {X 0,Y 305.383,Z 637.033,A -85,B 0,C 180,E1 -22210.65,E2 -22210.65} C_VEL
LIN {X 0,Y 310.706,Z 640.821,A -85,B 0,C 180,E1 -22211.799,E2 -22211.799} C_VEL
LIN {X 0,Y 316.848,Z 645.123,A -85,B 0,C 180,E1 -22213.241,E2 -22213.241} C_VEL
LIN {X 0,Y 322.816,Z 649.295,A -85,B 0,C 180,E1 -22214.856,E2 -22214.856} C_VEL
LIN {X 0,Y 327.952,Z 652.523,A -85,B 0,C 180,E1 -22216.366,E2 -22216.366} C_VEL
LIN {X 0,Y 332.203,Z 655.264,A -85,B 0,C 180,E1 -22217.787,E2 -22217.787} C_VEL
LIN {X 0,Y 336.055,Z 658.049,A -85,B 0,C 180,E1 -22219.381,E2 -22219.381} C_VEL
LIN {X 0,Y 338.417,Z 659.598,A -85,B 0,C 180,E1 -22220.437,E2 -22220.437} C_VEL
LIN {X 0,Y 340.972,Z 661.132,A -85,B 0,C 180,E1 -22221.704,E2 -22221.704} C_VEL
LIN {X 0,Y 343.229,Z 662.333,A -85,B 0,C 180,E1 -22222.943,E2 -22222.943} C_VEL
LIN {X 0,Y 345.839,Z 663.58,A -85,B 0,C 180,E1 -22224.694,E2 -22224.694} C_VEL
LIN {X 0,Y 347.971,Z 664.33,A -85,B 0,C 180,E1 -22226.526,E2 -22226.526} C_VEL
LIN {X 0,Y 348.767,Z 664.708,A -85,B 0,C 180,E1 -22227.69,E2 -22227.69} C_VEL
LIN {X 0,Y 349.178,Z 664.985,A -85,B 0,C 180,E1 -22228.847,E2 -22228.847} C_VEL
LIN {X 0,Y 349.465,Z 664.934,A -85,B 0,C 180,E1 -22230,E2 -22230} C_VEL
LIN {X 0,Y 349.199,Z 664.95,A -85,B 0,C 180,E1 -22231.153,E2 -22231.153} C_VEL
LIN {X 0,Y 348.741,Z 664.703,A -85,B 0,C 180,E1 -22232.31,E2 -22232.31} C_VEL
LIN {X 0,Y 347.95,Z 664.311,A -85,B 0,C 180,E1 -22233.474,E2 -22233.474} C_VEL
LIN {X 0,Y 345.847,Z 663.593,A -85,B 0,C 180,E1 -22235.322,E2 -22235.322} C_VEL
LIN {X 0,Y 343.168,Z 662.345,A -85,B 0,C 180,E1 -22237.058,E2 -22237.058} C_VEL
LIN {X 0,Y 340.905,Z 661.139,A -85,B 0,C 180,E1 -22238.306,E2 -22238.306} C_VEL
LIN {X 0,Y 338.384,Z 659.596,A -85,B 0,C 180,E1 -22239.564,E2 -22239.564} C_VEL
LIN {X 0,Y 335.464,Z 657.632,A -85,B 0,C 180,E1 -22240.868,E2 -22240.868} C_VEL
LIN {X 0,Y 331.221,Z 654.573,A -85,B 0,C 180,E1 -22242.577,E2 -22242.577} C_VEL
LIN {X 0,Y 325.24,Z 650.906,A -85,B 0,C 180,E1 -22244.441,E2 -22244.441} C_VEL
LIN {X 0,Y 318.53,Z 646.317,A -85,B 0,C 180,E1 -22246.318,E2 -22246.318} C_VEL
LIN {X 0,Y 313.303,Z 642.587,A -85,B 0,C 180,E1 -22247.635,E2 -22247.635} C_VEL
LIN {X 0,Y 305.407,Z 637.061,A -85,B 0,C 180,E1 -22249.362,E2 -22249.362} C_VEL
LIN {X 0,Y 298.818,Z 632.188,A -85,B 0,C 180,E1 -22250.658,E2 -22250.658} C_VEL
LIN {X 0,Y 284.678,Z 621.618,A -85,B 0,C 180,E1 -22253.138,E2 -22253.138} C_VEL
LIN {X 0,Y 272.191,Z 611.646,A -85,B 0,C 180,E1 -22255.358,E2 -22255.358} C_VEL
LIN {X 0,Y 259.305,Z 599.962,A -85,B 0,C 180,E1 -22257.744,E2 -22257.744} C_VEL
LIN {X 0,Y 247.799,Z 587.824,A -85,B 0,C 180,E1 -22259.917,E2 -22259.917} C_VEL
LIN {X 0,Y 236.445,Z 574.457,A -85,B 0,C 180,E1 -22262.047,E2 -22262.047} C_VEL
LIN {X 0,Y 226.621,Z 560.529,A -85,B 0,C 180,E1 -22264.149,E2 -22264.149} C_VEL
LIN {X 0,Y 219.156,Z 547.501,A -85,B 0,C 180,E1 -22266.011,E2 -22266.011} C_VEL
LIN {X 0,Y 209.606,Z 527.416,A -85,B 0,C 180,E1 -22268.808,E2 -22268.808} C_VEL
LIN {X 0,Y 202.917,Z 515.03,A -85,B 0,C 180,E1 -22270.922,E2 -22270.922} C_VEL
LIN {X 0,Y 195.851,Z 503.829,A -85,B 0,C 180,E1 -22273.305,E2 -22273.305} C_VEL
LIN {X 0,Y 191.274,Z 497.014,A -85,B 0,C 180,E1 -22274.974,E2 -22274.974} C_VEL
LIN {X 0,Y 189.023,Z 493.809,A -85,B 0,C 180,E1 -22275.837,E2 -22275.837} C_VEL
LIN {X 0,Y 188.132,Z 492.581,A -85,B 0,C 180,E1 -22276.185,E2 -22276.185} C_VEL
LIN {X 0,Y 186.355,Z 490.522,A -85,B 0,C 180,E1 -22276.876,E2 -22276.876} C_VEL
LIN {X 0,Y 185.541,Z 488.451,A -85,B 0,C 180,E1 -22277.412,E2 -22277.412} C_VEL
LIN {X 0,Y 185.445,Z 487.92,A -85,B 0,C 180,E1 -22277.931,E2 -22277.931} C_VEL
LIN {X 0,Y 185.491,Z 487.875,A -85,B 0,C 180,E1 -22282.717,E2 -22282.717} C_VEL
LIN {X 0,Y 185.521,Z 487.87,A -85,B 0,C 180,E1 -22287.975,E2 -22287.975} C_VEL
LIN {X 0,Y 185.482,Z 487.843,A -85,B 0,C 180,E1 -22292.959,E2 -22292.959} C_VEL
LIN {X 0,Y 185.539,Z 487.859,A -85,B 0,C 180,E1 -22297.745,E2 -22297.745} C_VEL
LIN {X 0,Y 185.632,Z 487.825,A -85,B 0,C 180,E1 -22302.373,E2 -22302.373} C_VEL
LIN {X 0,Y 185.702,Z 487.833,A -85,B 0,C 180,E1 -22306.879,E2 -22306.879} C_VEL
LIN {X 0,Y 185.968,Z 487.776,A -85,B 0,C 180,E1 -22311.309,E2 -22311.309} C_VEL
LIN {X 0,Y 186.161,Z 487.752,A -85,B 0,C 180,E1 -22317.84,E2 -22317.84} C_VEL
LIN {X 0,Y 186.373,Z 487.716,A -85,B 0,C 180,E1 -22320.003,E2 -22320.003} C_VEL
LIN {X 0,Y 185.876,Z 487.832,A -85,B 0,C 180,E1 -22324.34,E2 -22324.34} C_VEL
LIN {X 0,Y 185.968,Z 487.768,A -85,B 0,C 180,E1 -22328.698,E2 -22328.698} C_VEL
LIN {X 0,Y 185.683,Z 487.847,A -85,B 0,C 180,E1 -22333.129,E2 -22333.129} C_VEL
LIN {X 0,Y 185.62,Z 487.814,A -85,B 0,C 180,E1 -22338.818,E2 -22338.818} C_VEL
LIN {X 0,Y 185.545,Z 487.869,A -85,B 0,C 180,E1 -22342.261,E2 -22342.261} C_VEL
LIN {X 0,Y 185.493,Z 487.839,A -85,B 0,C 180,E1 -22347.046,E2 -22347.046} C_VEL
LIN {X 0,Y 185.533,Z 487.855,A -85,B 0,C 180,E1 -22352.031,E2 -22352.031} C_VEL
LIN {X 0,Y 185.504,Z 487.878,A -85,B 0,C 180,E1 -22357.317,E2 -22357.317} C_VEL
LIN {X 0,Y 185.487,Z 488.063,A -85,B 0,C 180,E1 -22360.32,E2 -22360.32} C_VEL
LIN {X 0,Y 186.162,Z 490.632,A -85,B 0,C 180,E1 -22362.499,E2 -22362.499} C_VEL
LIN {X 0,Y 187.761,Z 493.891,A -85,B 0,C 180,E1 -22363.378,E2 -22363.378} C_VEL
LIN {X 0,Y 189.879,Z 497.008,A -85,B 0,C 180,E1 -22364.211,E2 -22364.211} C_VEL
LIN {X 0,Y 195.898,Z 507.541,A -85,B 0,C 180,E1 -22366.503,E2 -22366.503} C_VEL
LIN {X 0,Y 200.941,Z 516.994,A -85,B 0,C 180,E1 -22368.287,E2 -22368.287} C_VEL
LIN {X 0,Y 207.432,Z 531.293,A -85,B 0,C 180,E1 -22370.485,E2 -22370.485} C_VEL
LIN {X 0,Y 210.637,Z 539.837,A -85,B 0,C 180,E1 -22371.56,E2 -22371.56} C_VEL
LIN {X 0,Y 212.753,Z 554.296,A -85,B 0,C 180,E1 -22372.61,E2 -22372.61} C_VEL
LIN {X 0,Y 210.444,Z 598.116,A -85,B 0,C 180,E1 -22374.038,E2 -22374.038} C_VEL
LIN {X 0,Y 209.416,Z 607.994,A -85,B 0,C 180,E1 -22374.554,E2 -22374.554} C_VEL
LIN {X 0,Y 207.984,Z 617.502,A -85,B 0,C 180,E1 -22375.235,E2 -22375.235} C_VEL
LIN {X 0,Y 206.343,Z 626.595,A -85,B 0,C 180,E1 -22376.102,E2 -22376.102} C_VEL
LIN {X 0,Y 204.263,Z 635.736,A -85,B 0,C 180,E1 -22377.187,E2 -22377.187} C_VEL
LIN {X 0,Y 201.952,Z 644.735,A -85,B 0,C 180,E1 -22378.534,E2 -22378.534} C_VEL
LIN {X 0,Y 199.408,Z 653.458,A -85,B 0,C 180,E1 -22380.144,E2 -22380.144} C_VEL
LIN {X 0,Y 197.058,Z 660.876,A -85,B 0,C 180,E1 -22381.8,E2 -22381.8} C_VEL
LIN {X 0,Y 193.989,Z 669.669,A -85,B 0,C 180,E1 -22384.231,E2 -22384.231} C_VEL
LIN {X 0,Y 191.963,Z 675.662,A -85,B 0,C 180,E1 -22386.252,E2 -22386.252} C_VEL
LIN {X 0,Y 189.608,Z 681.973,A -85,B 0,C 180,E1 -22388.815,E2 -22388.815} C_VEL
LIN {X 0,Y 187.596,Z 687.247,A -85,B 0,C 180,E1 -22391.432,E2 -22391.432} C_VEL
LIN {X 0,Y 185.587,Z 692.339,A -85,B 0,C 180,E1 -22394.628,E2 -22394.628} C_VEL
LIN {X 0,Y 185.181,Z 693.582,A -85,B 0,C 180,E1 -22395.572,E2 -22395.572} C_VEL
LIN {X 0,Y 183.882,Z 695.698,A -85,B 0,C 180,E1 -22397.242,E2 -22397.242} C_VEL
LIN {X 0,Y 180.18,Z 698.455,A -85,B 0,C 180,E1 -22400.007,E2 -22400.007} C_VEL
LIN {X 0,Y 177.302,Z 700.062,A -85,B 0,C 180,E1 -22402.335,E2 -22402.335} C_VEL
LIN {X 0,Y 176.074,Z 701.014,A -85,B 0,C 180,E1 -22404.195,E2 -22404.195} C_VEL
LIN {X 0,Y 175.963,Z 701.254,A -85,B 0,C 180,E1 -22404.832,E2 -22404.832} C_VEL
LIN {X 0,Y 175.957,Z 702.094,A -85,B 0,C 180,E1 -22407.711,E2 -22407.711} C_VEL
LIN {X 0,Y 176.061,Z 702.378,A -85,B 0,C 180,E1 -22410,E2 -22410} C_VEL
LIN {X 0,Y 175.955,Z 701.993,A -85,B 0,C 180,E1 -22413.034,E2 -22413.034} C_VEL
LIN {X 0,Y 176.122,Z 700.56,A -85,B 0,C 180,E1 -22416.875,E2 -22416.875} C_VEL
LIN {X 0,Y 177.001,Z 697.204,A -85,B 0,C 180,E1 -22421.451,E2 -22421.451} C_VEL
LIN {X 0,Y 178.199,Z 693.572,A -85,B 0,C 180,E1 -22424.854,E2 -22424.854} C_VEL
LIN {X 0,Y 180.08,Z 688.839,A -85,B 0,C 180,E1 -22428.193,E2 -22428.193} C_VEL
LIN {X 0,Y 182.498,Z 682.868,A -85,B 0,C 180,E1 -22431.459,E2 -22431.459} C_VEL
LIN {X 0,Y 184.705,Z 677.401,A -85,B 0,C 180,E1 -22433.86,E2 -22433.86} C_VEL
LIN {X 0,Y 187.069,Z 671.034,A -85,B 0,C 180,E1 -22436.195,E2 -22436.195} C_VEL
LIN {X 0,Y 189.476,Z 664.379,A -85,B 0,C 180,E1 -22438.224,E2 -22438.224} C_VEL
LIN {X 0,Y 192.173,Z 656.554,A -85,B 0,C 180,E1 -22440.189,E2 -22440.189} C_VEL
LIN {X 0,Y 194.806,Z 648.476,A -85,B 0,C 180,E1 -22441.845,E2 -22441.845} C_VEL
LIN {X 0,Y 197.541,Z 638.719,A -85,B 0,C 180,E1 -22443.466,E2 -22443.466} C_VEL
LIN {X 0,Y 199.601,Z 630.333,A -85,B 0,C 180,E1 -22444.594,E2 -22444.594} C_VEL
LIN {X 0,Y 201.727,Z 619.829,A -85,B 0,C 180,E1 -22445.701,E2 -22445.701} C_VEL
LIN {X 0,Y 203.468,Z 609.399,A -85,B 0,C 180,E1 -22446.504,E2 -22446.504} C_VEL
LIN {X 0,Y 204.704,Z 599.052,A -85,B 0,C 180,E1 -22447.067,E2 -22447.067} C_VEL
LIN {X 0,Y 205.913,Z 577.566,A -85,B 0,C 180,E1 -22447.837,E2 -22447.837} C_VEL
LIN {X 0,Y 207.001,Z 554.447,A -85,B 0,C 180,E1 -22448.601,E2 -22448.601} C_VEL
LIN {X 0,Y 204.904,Z 541.158,A -85,B 0,C 180,E1 -22449.656,E2 -22449.656} C_VEL
LIN {X 0,Y 199.684,Z 528.423,A -85,B 0,C 180,E1 -22451.495,E2 -22451.495} C_VEL
LIN {X 0,Y 194.676,Z 517.784,A -85,B 0,C 180,E1 -22453.328,E2 -22453.328} C_VEL
LIN {X 0,Y 187.732,Z 505.153,A -85,B 0,C 180,E1 -22456.022,E2 -22456.022} C_VEL
LIN {X 0,Y 184.636,Z 500.008,A -85,B 0,C 180,E1 -22457.307,E2 -22457.307} C_VEL
LIN {X 0,Y 181.674,Z 495.242,A -85,B 0,C 180,E1 -22458.6,E2 -22458.6} C_VEL
LIN {X 0,Y 179.212,Z 491.38,A -85,B 0,C 180,E1 -22459.768,E2 -22459.768} C_VEL
LIN {X 0,Y 178.709,Z 490.146,A -85,B 0,C 180,E1 -22460.275,E2 -22460.275} C_VEL
LIN {X 0,Y 178.404,Z 488.83,A -85,B 0,C 180,E1 -22461.547,E2 -22461.547} C_VEL
LIN {X 0,Y 178.487,Z 488.721,A -85,B 0,C 180,E1 -22466.543,E2 -22466.543} C_VEL
LIN {X 0,Y 178.425,Z 488.727,A -85,B 0,C 180,E1 -22471.789,E2 -22471.789} C_VEL
LIN {X 0,Y 178.465,Z 488.75,A -85,B 0,C 180,E1 -22476.805,E2 -22476.805} C_VEL
LIN {X 0,Y 178.597,Z 488.688,A -85,B 0,C 180,E1 -22481.647,E2 -22481.647} C_VEL
LIN {X 0,Y 178.613,Z 488.732,A -85,B 0,C 180,E1 -22486.341,E2 -22486.341} C_VEL
LIN {X 0,Y 178.9,Z 488.646,A -85,B 0,C 180,E1 -22490.956,E2 -22490.956} C_VEL
LIN {X 0,Y 179.118,Z 488.643,A -85,B 0,C 180,E1 -22497.748,E2 -22497.748} C_VEL
LIN {X 0,Y 179.339,Z 488.592,A -85,B 0,C 180,E1 -22499.997,E2 -22499.997} C_VEL
LIN {X 0,Y 178.888,Z 488.688,A -85,B 0,C 180,E1 -22506.765,E2 -22506.765} C_VEL
LIN {X 0,Y 178.829,Z 488.658,A -85,B 0,C 180,E1 -22510.738,E2 -22510.738} C_VEL
LIN {X 0,Y 178.566,Z 488.731,A -85,B 0,C 180,E1 -22515.988,E2 -22515.988} C_VEL
LIN {X 0,Y 178.549,Z 488.697,A -85,B 0,C 180,E1 -22519.148,E2 -22519.148} C_VEL
LIN {X 0,Y 178.457,Z 488.736,A -85,B 0,C 180,E1 -22525.072,E2 -22525.072} C_VEL
LIN {X 0,Y 178.442,Z 488.756,A -85,B 0,C 180,E1 -22530.793,E2 -22530.793} C_VEL
LIN {X 0,Y 178.473,Z 488.724,A -85,B 0,C 180,E1 -22534.215,E2 -22534.215} C_VEL
LIN {X 0,Y 178.435,Z 488.938,A -85,B 0,C 180,E1 -22539.789,E2 -22539.789} C_VEL
LIN {X 0,Y 178.628,Z 489.773,A -85,B 0,C 180,E1 -22540.29,E2 -22540.29} C_VEL
LIN {X 0,Y 180.199,Z 492.661,A -85,B 0,C 180,E1 -22541.104,E2 -22541.104} C_VEL
LIN {X 0,Y 181.868,Z 494.244,A -85,B 0,C 180,E1 -22541.8,E2 -22541.8} C_VEL
LIN {X 0,Y 184.061,Z 497.653,A -85,B 0,C 180,E1 -22542.756,E2 -22542.756} C_VEL
LIN {X 0,Y 185.542,Z 499.604,A -85,B 0,C 180,E1 -22543.36,E2 -22543.36} C_VEL
LIN {X 0,Y 191.609,Z 508.497,A -85,B 0,C 180,E1 -22545.72,E2 -22545.72} C_VEL
LIN {X 0,Y 197.911,Z 518.649,A -85,B 0,C 180,E1 -22547.974,E2 -22547.974} C_VEL
LIN {X 0,Y 203.617,Z 529.093,A -85,B 0,C 180,E1 -22549.89,E2 -22549.89} C_VEL
LIN {X 0,Y 209.275,Z 540.945,A -85,B 0,C 180,E1 -22551.702,E2 -22551.702} C_VEL
LIN {X 0,Y 216.553,Z 556.075,A -85,B 0,C 180,E1 -22553.83,E2 -22553.83} C_VEL
LIN {X 0,Y 224.797,Z 569.545,A -85,B 0,C 180,E1 -22555.874,E2 -22555.874} C_VEL
LIN {X 0,Y 233.467,Z 581.437,A -85,B 0,C 180,E1 -22557.741,E2 -22557.741} C_VEL
LIN {X 0,Y 243.8,Z 593.685,A -85,B 0,C 180,E1 -22559.854,E2 -22559.854} C_VEL
LIN {X 0,Y 254.496,Z 605.127,A -85,B 0,C 180,E1 -22562.084,E2 -22562.084} C_VEL
LIN {X 0,Y 266.623,Z 616.238,A -85,B 0,C 180,E1 -22564.522,E2 -22564.522} C_VEL
LIN {X 0,Y 279.965,Z 626.84,A -85,B 0,C 180,E1 -22567.063,E2 -22567.063} C_VEL
LIN {X 0,Y 292.727,Z 636.256,A -85,B 0,C 180,E1 -22569.437,E2 -22569.437} C_VEL
LIN {X 0,Y 300.101,Z 641.641,A -85,B 0,C 180,E1 -22570.861,E2 -22570.861} C_VEL
LIN {X 0,Y 307.399,Z 646.812,A -85,B 0,C 180,E1 -22572.425,E2 -22572.425} C_VEL
LIN {X 0,Y 314.195,Z 651.643,A -85,B 0,C 180,E1 -22574.11,E2 -22574.11} C_VEL
LIN {X 0,Y 321.158,Z 656.228,A -85,B 0,C 180,E1 -22576.071,E2 -22576.071} C_VEL
LIN {X 0,Y 325.801,Z 659.119,A -85,B 0,C 180,E1 -22577.543,E2 -22577.543} C_VEL
LIN {X 0,Y 331.092,Z 662.919,A -85,B 0,C 180,E1 -22579.675,E2 -22579.675} C_VEL
LIN {X 0,Y 335.101,Z 665.42,A -85,B 0,C 180,E1 -22581.558,E2 -22581.558} C_VEL
LIN {X 0,Y 337.428,Z 666.719,A -85,B 0,C 180,E1 -22582.821,E2 -22582.821} C_VEL
LIN {X 0,Y 339.412,Z 667.716,A -85,B 0,C 180,E1 -22584.057,E2 -22584.057} C_VEL
LIN {X 0,Y 341.093,Z 668.44,A -85,B 0,C 180,E1 -22585.273,E2 -22585.273} C_VEL
LIN {X 0,Y 342.462,Z 668.907,A -85,B 0,C 180,E1 -22586.47,E2 -22586.47} C_VEL
LIN {X 0,Y 343.316,Z 669.287,A -85,B 0,C 180,E1 -22587.654,E2 -22587.654} C_VEL
LIN {X 0,Y 343.761,Z 669.556,A -85,B 0,C 180,E1 -22588.829,E2 -22588.829} C_VEL
LIN {X 0,Y 344.051,Z 669.525,A -85,B 0,C 180,E1 -22590,E2 -22590} C_VEL
LIN {X 0,Y 343.782,Z 669.525,A -85,B 0,C 180,E1 -22591.171,E2 -22591.171} C_VEL
LIN {X 0,Y 343.306,Z 669.27,A -85,B 0,C 180,E1 -22592.346,E2 -22592.346} C_VEL
LIN {X 0,Y 342.441,Z 668.89,A -85,B 0,C 180,E1 -22593.53,E2 -22593.53} C_VEL
LIN {X 0,Y 341.069,Z 668.418,A -85,B 0,C 180,E1 -22594.728,E2 -22594.728} C_VEL
LIN {X 0,Y 339.218,Z 667.625,A -85,B 0,C 180,E1 -22596.05,E2 -22596.05} C_VEL
LIN {X 0,Y 337.383,Z 666.724,A -85,B 0,C 180,E1 -22597.18,E2 -22597.18} C_VEL
LIN {X 0,Y 334.268,Z 664.995,A -85,B 0,C 180,E1 -22598.836,E2 -22598.836} C_VEL
LIN {X 0,Y 331.108,Z 662.925,A -85,B 0,C 180,E1 -22600.318,E2 -22600.318} C_VEL
LIN {X 0,Y 325.801,Z 659.109,A -85,B 0,C 180,E1 -22602.457,E2 -22602.457} C_VEL
LIN {X 0,Y 319.321,Z 655.132,A -85,B 0,C 180,E1 -22604.452,E2 -22604.452} C_VEL
LIN {X 0,Y 314.198,Z 651.627,A -85,B 0,C 180,E1 -22605.892,E2 -22605.892} C_VEL
LIN {X 0,Y 307.444,Z 646.847,A -85,B 0,C 180,E1 -22607.572,E2 -22607.572} C_VEL
LIN {X 0,Y 300.231,Z 641.731,A -85,B 0,C 180,E1 -22609.13,E2 -22609.13} C_VEL
LIN {X 0,Y 292.737,Z 636.218,A -85,B 0,C 180,E1 -22610.568,E2 -22610.568} C_VEL
LIN {X 0,Y 281.673,Z 628.079,A -85,B 0,C 180,E1 -22612.611,E2 -22612.611} C_VEL
LIN {X 0,Y 269.352,Z 618.471,A -85,B 0,C 180,E1 -22614.953,E2 -22614.953} C_VEL
LIN {X 0,Y 258.535,Z 608.925,A -85,B 0,C 180,E1 -22617.099,E2 -22617.099} C_VEL
LIN {X 0,Y 249.35,Z 599.703,A -85,B 0,C 180,E1 -22618.996,E2 -22618.996} C_VEL
LIN {X 0,Y 239.078,Z 588.282,A -85,B 0,C 180,E1 -22621.118,E2 -22621.118} C_VEL
LIN {X 0,Y 228.371,Z 574.764,A -85,B 0,C 180,E1 -22623.322,E2 -22623.322} C_VEL
LIN {X 0,Y 219.203,Z 560.696,A -85,B 0,C 180,E1 -22625.479,E2 -22625.479} C_VEL
LIN {X 0,Y 212.111,Z 547.289,A -85,B 0,C 180,E1 -22627.425,E2 -22627.425} C_VEL
LIN {X 0,Y 204.596,Z 531.014,A -85,B 0,C 180,E1 -22629.792,E2 -22629.792} C_VEL
LIN {X 0,Y 198.277,Z 519.23,A -85,B 0,C 180,E1 -22631.902,E2 -22631.902} C_VEL
LIN {X 0,Y 190.972,Z 507.441,A -85,B 0,C 180,E1 -22634.523,E2 -22634.523} C_VEL
LIN {X 0,Y 186.883,Z 501.58,A -85,B 0,C 180,E1 -22636.096,E2 -22636.096} C_VEL
LIN {X 0,Y 184.467,Z 498.097,A -85,B 0,C 180,E1 -22637.082,E2 -22637.082} C_VEL
LIN {X 0,Y 182.238,Z 494.992,A -85,B 0,C 180,E1 -22638.026,E2 -22638.026} C_VEL
LIN {X 0,Y 181.535,Z 493.818,A -85,B 0,C 180,E1 -22638.344,E2 -22638.344} C_VEL
LIN {X 0,Y 179.436,Z 491.61,A -85,B 0,C 180,E1 -22639.241,E2 -22639.241} C_VEL
LIN {X 0,Y 178.517,Z 489.4,A -85,B 0,C 180,E1 -22639.865,E2 -22639.865} C_VEL
LIN {X 0,Y 178.397,Z 488.796,A -85,B 0,C 180,E1 -22640.567,E2 -22640.567} C_VEL
LIN {X 0,Y 178.473,Z 488.724,A -85,B 0,C 180,E1 -22645.785,E2 -22645.785} C_VEL
LIN {X 0,Y 178.456,Z 488.738,A -85,B 0,C 180,E1 -22650.043,E2 -22650.043} C_VEL
LIN {X 0,Y 178.457,Z 488.736,A -85,B 0,C 180,E1 -22654.928,E2 -22654.928} C_VEL
LIN {X 0,Y 178.549,Z 488.697,A -85,B 0,C 180,E1 -22660.852,E2 -22660.852} C_VEL
LIN {X 0,Y 178.627,Z 488.723,A -85,B 0,C 180,E1 -22666.349,E2 -22666.349} C_VEL
LIN {X 0,Y 178.899,Z 488.652,A -85,B 0,C 180,E1 -22670.963,E2 -22670.963} C_VEL
LIN {X 0,Y 178.824,Z 488.705,A -85,B 0,C 180,E1 -22675.495,E2 -22675.495} C_VEL
LIN {X 0,Y 179.339,Z 488.592,A -85,B 0,C 180,E1 -22680.003,E2 -22680.003} C_VEL
LIN {X 0,Y 178.825,Z 488.71,A -85,B 0,C 180,E1 -22684.512,E2 -22684.512} C_VEL
LIN {X 0,Y 178.9,Z 488.646,A -85,B 0,C 180,E1 -22689.044,E2 -22689.044} C_VEL
LIN {X 0,Y 178.613,Z 488.732,A -85,B 0,C 180,E1 -22693.659,E2 -22693.659} C_VEL
LIN {X 0,Y 178.551,Z 488.696,A -85,B 0,C 180,E1 -22699.15,E2 -22699.15} C_VEL
LIN {X 0,Y 178.466,Z 488.721,A -85,B 0,C 180,E1 -22705.078,E2 -22705.078} C_VEL
LIN {X 0,Y 178.453,Z 488.755,A -85,B 0,C 180,E1 -22710.799,E2 -22710.799} C_VEL
LIN {X 0,Y 178.486,Z 488.721,A -85,B 0,C 180,E1 -22714.22,E2 -22714.22} C_VEL
LIN {X 0,Y 178.409,Z 488.818,A -85,B 0,C 180,E1 -22718.451,E2 -22718.451} C_VEL
LIN {X 0,Y 178.809,Z 490.401,A -85,B 0,C 180,E1 -22719.882,E2 -22719.882} C_VEL
LIN {X 0,Y 180.969,Z 494.342,A -85,B 0,C 180,E1 -22721.095,E2 -22721.095} C_VEL
LIN {X 0,Y 182.832,Z 496.996,A -85,B 0,C 180,E1 -22721.908,E2 -22721.908} C_VEL
LIN {X 0,Y 186.36,Z 502.836,A -85,B 0,C 180,E1 -22723.416,E2 -22723.416} C_VEL
LIN {X 0,Y 191.146,Z 511.227,A -85,B 0,C 180,E1 -22725.336,E2 -22725.336} C_VEL
LIN {X 0,Y 196.914,Z 522.341,A -85,B 0,C 180,E1 -22727.5,E2 -22727.5} C_VEL
LIN {X 0,Y 202.623,Z 535.335,A -85,B 0,C 180,E1 -22729.547,E2 -22729.547} C_VEL
LIN {X 0,Y 205.346,Z 542.793,A -85,B 0,C 180,E1 -22730.518,E2 -22730.518} C_VEL
LIN {X 0,Y 207.086,Z 555.354,A -85,B 0,C 180,E1 -22731.457,E2 -22731.457} C_VEL
LIN {X 0,Y 204.786,Z 597.328,A -85,B 0,C 180,E1 -22732.844,E2 -22732.844} C_VEL
LIN {X 0,Y 203.715,Z 607.575,A -85,B 0,C 180,E1 -22733.385,E2 -22733.385} C_VEL
LIN {X 0,Y 202.205,Z 617.306,A -85,B 0,C 180,E1 -22734.09,E2 -22734.09} C_VEL
LIN {X 0,Y 200.48,Z 626.398,A -85,B 0,C 180,E1 -22734.968,E2 -22734.968} C_VEL
LIN {X 0,Y 198.33,Z 635.54,A -85,B 0,C 180,E1 -22736.075,E2 -22736.075} C_VEL
LIN {X 0,Y 195.921,Z 644.538,A -85,B 0,C 180,E1 -22737.448,E2 -22737.448} C_VEL
LIN {X 0,Y 193.27,Z 653.261,A -85,B 0,C 180,E1 -22739.094,E2 -22739.094} C_VEL
LIN {X 0,Y 190.821,Z 660.68,A -85,B 0,C 180,E1 -22740.791,E2 -22740.791} C_VEL
LIN {X 0,Y 187.591,Z 669.472,A -85,B 0,C 180,E1 -22743.284,E2 -22743.284} C_VEL
LIN {X 0,Y 185.175,Z 676.142,A -85,B 0,C 180,E1 -22745.633,E2 -22745.633} C_VEL
LIN {X 0,Y 183.006,Z 681.777,A -85,B 0,C 180,E1 -22748.011,E2 -22748.011} C_VEL
LIN {X 0,Y 180.858,Z 687.05,A -85,B 0,C 180,E1 -22750.713,E2 -22750.713} C_VEL
LIN {X 0,Y 178.719,Z 692.142,A -85,B 0,C 180,E1 -22754.022,E2 -22754.022} C_VEL
LIN {X 0,Y 177.355,Z 696.113,A -85,B 0,C 180,E1 -22757.412,E2 -22757.412} C_VEL
LIN {X 0,Y 176.464,Z 699.054,A -85,B 0,C 180,E1 -22760.833,E2 -22760.833} C_VEL
LIN {X 0,Y 176.094,Z 700.559,A -85,B 0,C 180,E1 -22763.123,E2 -22763.123} C_VEL
LIN {X 0,Y 175.963,Z 701.254,A -85,B 0,C 180,E1 -22764.832,E2 -22764.832} C_VEL
LIN {X 0,Y 175.247,Z 701.941,A -85,B 0,C 180,E1 -22766.733,E2 -22766.733} C_VEL
LIN {X 0,Y 173.639,Z 702.218,A -85,B 0,C 180,E1 -22768.612,E2 -22768.612} C_VEL
LIN {X 0,Y 169.938,Z 701.975,A -85,B 0,C 180,E1 -22772.432,E2 -22772.432} C_VEL
LIN {X 0,Y 168.94,Z 701.442,A -85,B 0,C 180,E1 -22774.426,E2 -22774.426} C_VEL
LIN {X 0,Y 168.877,Z 701.169,A -85,B 0,C 180,E1 -22775.1,E2 -22775.1} C_VEL
LIN {X 0,Y 169.047,Z 700.363,A -85,B 0,C 180,E1 -22777.165,E2 -22777.165} C_VEL
LIN {X 0,Y 170.028,Z 697.007,A -85,B 0,C 180,E1 -22781.927,E2 -22781.927} C_VEL
LIN {X 0,Y 171.306,Z 693.374,A -85,B 0,C 180,E1 -22785.466,E2 -22785.466} C_VEL
LIN {X 0,Y 173.332,Z 688.643,A -85,B 0,C 180,E1 -22788.927,E2 -22788.927} C_VEL
LIN {X 0,Y 175.402,Z 683.763,A -85,B 0,C 180,E1 -22791.754,E2 -22791.754} C_VEL
LIN {X 0,Y 177.917,Z 677.893,A -85,B 0,C 180,E1 -22794.504,E2 -22794.504} C_VEL
LIN {X 0,Y 180.118,Z 672.398,A -85,B 0,C 180,E1 -22796.661,E2 -22796.661} C_VEL
LIN {X 0,Y 183.235,Z 664.182,A -85,B 0,C 180,E1 -22799.276,E2 -22799.276} C_VEL
LIN {X 0,Y 186.067,Z 656.358,A -85,B 0,C 180,E1 -22801.289,E2 -22801.289} C_VEL
LIN {X 0,Y 188.82,Z 648.28,A -85,B 0,C 180,E1 -22802.98,E2 -22802.98} C_VEL
LIN {X 0,Y 191.647,Z 638.523,A -85,B 0,C 180,E1 -22804.639,E2 -22804.639} C_VEL
LIN {X 0,Y 193.791,Z 630.136,A -85,B 0,C 180,E1 -22805.787,E2 -22805.787} C_VEL
LIN {X 0,Y 196.011,Z 619.633,A -85,B 0,C 180,E1 -22806.91,E2 -22806.91} C_VEL
LIN {X 0,Y 197.84,Z 608.974,A -85,B 0,C 180,E1 -22807.741,E2 -22807.741} C_VEL
LIN {X 0,Y 199.129,Z 598.42,A -85,B 0,C 180,E1 -22808.315,E2 -22808.315} C_VEL
LIN {X 0,Y 200.437,Z 575.811,A -85,B 0,C 180,E1 -22809.134,E2 -22809.134} C_VEL
LIN {X 0,Y 201.4,Z 555.066,A -85,B 0,C 180,E1 -22809.848,E2 -22809.848} C_VEL
LIN {X 0,Y 199.672,Z 544.069,A -85,B 0,C 180,E1 -22810.768,E2 -22810.768} C_VEL
LIN {X 0,Y 194.809,Z 532.061,A -85,B 0,C 180,E1 -22812.589,E2 -22812.589} C_VEL
LIN {X 0,Y 190.211,Z 522.079,A -85,B 0,C 180,E1 -22814.379,E2 -22814.379} C_VEL
LIN {X 0,Y 183.736,Z 510.002,A -85,B 0,C 180,E1 -22817.048,E2 -22817.048} C_VEL
LIN {X 0,Y 180.524,Z 504.571,A -85,B 0,C 180,E1 -22818.464,E2 -22818.464} C_VEL
LIN {X 0,Y 177.874,Z 500.256,A -85,B 0,C 180,E1 -22819.692,E2 -22819.692} C_VEL
LIN {X 0,Y 174.6,Z 495.203,A -85,B 0,C 180,E1 -22821.289,E2 -22821.289} C_VEL
LIN {X 0,Y 171.951,Z 491.703,A -85,B 0,C 180,E1 -22822.645,E2 -22822.645} C_VEL
LIN {X 0,Y 171.473,Z 490.201,A -85,B 0,C 180,E1 -22823.168,E2 -22823.168} C_VEL
LIN {X 0,Y 171.403,Z 489.683,A -85,B 0,C 180,E1 -22823.881,E2 -22823.881} C_VEL
LIN {X 0,Y 171.409,Z 489.635,A -85,B 0,C 180,E1 -22829.431,E2 -22829.431} C_VEL
LIN {X 0,Y 171.404,Z 489.596,A -85,B 0,C 180,E1 -22834.429,E2 -22834.429} C_VEL
LIN {X 0,Y 171.476,Z 489.578,A -85,B 0,C 180,E1 -22840.502,E2 -22840.502} C_VEL
LIN {X 0,Y 171.529,Z 489.615,A -85,B 0,C 180,E1 -22845.765,E2 -22845.765} C_VEL
LIN {X 0,Y 171.84,Z 489.524,A -85,B 0,C 180,E1 -22850.581,E2 -22850.581} C_VEL
LIN {X 0,Y 171.775,Z 489.588,A -85,B 0,C 180,E1 -22855.303,E2 -22855.303} C_VEL
LIN {X 0,Y 172.303,Z 489.467,A -85,B 0,C 180,E1 -22859.996,E2 -22859.996} C_VEL
LIN {X 0,Y 171.851,Z 489.556,A -85,B 0,C 180,E1 -22867.044,E2 -22867.044} C_VEL
LIN {X 0,Y 171.763,Z 489.538,A -85,B 0,C 180,E1 -22870.889,E2 -22870.889} C_VEL
LIN {X 0,Y 171.499,Z 489.597,A -85,B 0,C 180,E1 -22876.666,E2 -22876.666} C_VEL
LIN {X 0,Y 171.473,Z 489.578,A -85,B 0,C 180,E1 -22879.495,E2 -22879.495} C_VEL
LIN {X 0,Y 171.394,Z 489.608,A -85,B 0,C 180,E1 -22885.565,E2 -22885.565} C_VEL
LIN {X 0,Y 171.397,Z 489.627,A -85,B 0,C 180,E1 -22890.562,E2 -22890.562} C_VEL
